LIN {X 0,Y 538.14,Z 616.393,A -85,B 0,C 180,E1 -4151.68,E2 -4151.68} C_VEL
LIN {X 0,Y 538.436,Z 594.869,A -85,B 0,C 180,E1 -4154.665,E2 -4154.665} C_VEL
LIN {X 0,Y 538.828,Z 571.509,A -85,B 0,C 180,E1 -4157.948,E2 -4157.948} C_VEL
LIN {X 0,Y 539.184,Z 551.118,A -85,B 0,C 180,E1 -4160.805,E2 -4160.805} C_VEL
LIN {X 0,Y 539.601,Z 529.757,A -85,B 0,C 180,E1 -4163.813,E2 -4163.813} C_VEL
LIN {X 0,Y 539.337,Z 523.937,A -85,B 0,C 180,E1 -4164.645,E2 -4164.645} C_VEL
LIN {X 0,Y 539.061,Z 522.492,A -85,B 0,C 180,E1 -4164.86,E2 -4164.86} C_VEL
LIN {X 0,Y 537.997,Z 520.573,A -85,B 0,C 180,E1 -4165.217,E2 -4165.217} C_VEL
LIN {X 0,Y 535.449,Z 519.098,A -85,B 0,C 180,E1 -4165.705,E2 -4165.705} C_VEL
LIN {X 0,Y 532.19,Z 518.422,A -85,B 0,C 180,E1 -4166.352,E2 -4166.352} C_VEL
LIN {X 0,Y 531.093,Z 518.344,A -85,B 0,C 180,E1 -4166.774,E2 -4166.774} C_VEL
LIN {X 0,Y 531.002,Z 518.341,A -85,B 0,C 180,E1 -4166.921,E2 -4166.921} C_VEL
LIN {X 0,Y 530.985,Z 518.344,A -85,B 0,C 180,E1 -4169.323,E2 -4169.323} C_VEL
LIN {X 0,Y 530.969,Z 518.345,A -85,B 0,C 180,E1 -4172.1,E2 -4172.1} C_VEL
LIN {X 0,Y 530.987,Z 518.339,A -85,B 0,C 180,E1 -4174.853,E2 -4174.853} C_VEL
LIN {X 0,Y 530.969,Z 518.349,A -85,B 0,C 180,E1 -4177.508,E2 -4177.508} C_VEL
LIN {X 0,Y 530.985,Z 518.333,A -85,B 0,C 180,E1 -4180.433,E2 -4180.433} C_VEL
LIN {X 0,Y 530.952,Z 518.337,A -85,B 0,C 180,E1 -4183.279,E2 -4183.279} C_VEL
LIN {X 0,Y 530.986,Z 518.344,A -85,B 0,C 180,E1 -4185.621,E2 -4185.621} C_VEL
LIN {X 0,Y 530.998,Z 518.336,A -85,B 0,C 180,E1 -4188.564,E2 -4188.564} C_VEL
LIN {X 0,Y 530.961,Z 518.344,A -85,B 0,C 180,E1 -4191.529,E2 -4191.529} C_VEL
LIN {X 0,Y 530.958,Z 518.342,A -85,B 0,C 180,E1 -4194.38,E2 -4194.38} C_VEL
LIN {X 0,Y 530.971,Z 518.349,A -85,B 0,C 180,E1 -4197.133,E2 -4197.133} C_VEL
LIN {X 0,Y 530.974,Z 518.341,A -85,B 0,C 180,E1 -4199.803,E2 -4199.803} C_VEL
LIN {X 0,Y 531.018,Z 518.338,A -85,B 0,C 180,E1 -4202.467,E2 -4202.467} C_VEL
LIN {X 0,Y 530.999,Z 518.342,A -85,B 0,C 180,E1 -4204.942,E2 -4204.942} C_VEL
LIN {X 0,Y 530.977,Z 518.342,A -85,B 0,C 180,E1 -4208.246,E2 -4208.246} C_VEL
LIN {X 0,Y 531.049,Z 518.493,A -85,B 0,C 180,E1 -4209.545,E2 -4209.545} C_VEL
LIN {X 0,Y 531.712,Z 523.2,A -85,B 0,C 180,E1 -4210.505,E2 -4210.505} C_VEL
LIN {X 0,Y 531.398,Z 538.775,A -85,B 0,C 180,E1 -4213.48,E2 -4213.48} C_VEL
LIN {X 0,Y 531.21,Z 547.447,A -85,B 0,C 180,E1 -4215.07,E2 -4215.07} C_VEL
LIN {X 0,Y 531.552,Z 549.947,A -85,B 0,C 180,E1 -4215.153,E2 -4215.153} C_VEL
LIN {X 0,Y 532.79,Z 556.751,A -85,B 0,C 180,E1 -4215.282,E2 -4215.282} C_VEL
LIN {X 0,Y 532.431,Z 654.189,A -85,B 0,C 180,E1 -4216.619,E2 -4216.619} C_VEL
LIN {X 0,Y 532.263,Z 667.4,A -85,B 0,C 180,E1 -4216.955,E2 -4216.955} C_VEL
LIN {X 0,Y 532.009,Z 679.509,A -85,B 0,C 180,E1 -4217.41,E2 -4217.41} C_VEL
LIN {X 0,Y 531.827,Z 691.229,A -85,B 0,C 180,E1 -4218.006,E2 -4218.006} C_VEL
LIN {X 0,Y 531.56,Z 702.618,A -85,B 0,C 180,E1 -4218.754,E2 -4218.754} C_VEL
LIN {X 0,Y 531.28,Z 713.098,A -85,B 0,C 180,E1 -4219.616,E2 -4219.616} C_VEL
LIN {X 0,Y 531.071,Z 721.693,A -85,B 0,C 180,E1 -4220.478,E2 -4220.478} C_VEL
LIN {X 0,Y 530.892,Z 729.61,A -85,B 0,C 180,E1 -4221.435,E2 -4221.435} C_VEL
LIN {X 0,Y 530.69,Z 737.354,A -85,B 0,C 180,E1 -4222.581,E2 -4222.581} C_VEL
LIN {X 0,Y 530.607,Z 744.464,A -85,B 0,C 180,E1 -4223.917,E2 -4223.917} C_VEL
LIN {X 0,Y 530.459,Z 749.203,A -85,B 0,C 180,E1 -4225.059,E2 -4225.059} C_VEL
LIN {X 0,Y 530.516,Z 752.832,A -85,B 0,C 180,E1 -4226.201,E2 -4226.201} C_VEL
LIN {X 0,Y 530.457,Z 754.711,A -85,B 0,C 180,E1 -4226.962,E2 -4226.962} C_VEL
LIN {X 0,Y 530.411,Z 756.13,A -85,B 0,C 180,E1 -4227.721,E2 -4227.721} C_VEL
LIN {X 0,Y 530.344,Z 757.757,A -85,B 0,C 180,E1 -4229.24,E2 -4229.24} C_VEL
LIN {X 0,Y 530.343,Z 757.996,A -85,B 0,C 180,E1 -4229.999,E2 -4229.999} C_VEL
LIN {X 0,Y 530.344,Z 757.814,A -85,B 0,C 180,E1 -4230.759,E2 -4230.759} C_VEL
LIN {X 0,Y 530.411,Z 756.265,A -85,B 0,C 180,E1 -4232.277,E2 -4232.277} C_VEL
LIN {X 0,Y 530.457,Z 754.903,A -85,B 0,C 180,E1 -4233.037,E2 -4233.037} C_VEL
LIN {X 0,Y 530.523,Z 752.021,A -85,B 0,C 180,E1 -4234.178,E2 -4234.178} C_VEL
LIN {X 0,Y 530.523,Z 748.12,A -85,B 0,C 180,E1 -4235.32,E2 -4235.32} C_VEL
LIN {X 0,Y 530.592,Z 742.537,A -85,B 0,C 180,E1 -4236.575,E2 -4236.575} C_VEL
LIN {X 0,Y 530.758,Z 735.529,A -85,B 0,C 180,E1 -4237.8,E2 -4237.8} C_VEL
LIN {X 0,Y 530.927,Z 727.343,A -85,B 0,C 180,E1 -4238.947,E2 -4238.947} C_VEL
LIN {X 0,Y 531.104,Z 718.972,A -85,B 0,C 180,E1 -4239.905,E2 -4239.905} C_VEL
LIN {X 0,Y 531.418,Z 708.669,A -85,B 0,C 180,E1 -4240.862,E2 -4240.862} C_VEL
LIN {X 0,Y 531.692,Z 698.123,A -85,B 0,C 180,E1 -4241.651,E2 -4241.651} C_VEL
LIN {X 0,Y 531.871,Z 687.285,A -85,B 0,C 180,E1 -4242.302,E2 -4242.302} C_VEL
LIN {X 0,Y 532.16,Z 674.779,A -85,B 0,C 180,E1 -4242.876,E2 -4242.876} C_VEL
LIN {X 0,Y 532.357,Z 661.342,A -85,B 0,C 180,E1 -4243.308,E2 -4243.308} C_VEL
LIN {X 0,Y 532.508,Z 647.991,A -85,B 0,C 180,E1 -4243.572,E2 -4243.572} C_VEL
LIN {X 0,Y 532.735,Z 556.433,A -85,B 0,C 180,E1 -4244.814,E2 -4244.814} C_VEL
LIN {X 0,Y 531.26,Z 547.806,A -85,B 0,C 180,E1 -4244.989,E2 -4244.989} C_VEL
LIN {X 0,Y 531.226,Z 545.512,A -85,B 0,C 180,E1 -4245.342,E2 -4245.342} C_VEL
LIN {X 0,Y 531.549,Z 530.014,A -85,B 0,C 180,E1 -4248.281,E2 -4248.281} C_VEL
LIN {X 0,Y 531.675,Z 522.634,A -85,B 0,C 180,E1 -4249.698,E2 -4249.698} C_VEL
LIN {X 0,Y 531.04,Z 518.404,A -85,B 0,C 180,E1 -4250.58,E2 -4250.58} C_VEL
LIN {X 0,Y 530.998,Z 518.339,A -85,B 0,C 180,E1 -4254.042,E2 -4254.042} C_VEL
LIN {X 0,Y 531.006,Z 518.336,A -85,B 0,C 180,E1 -4256.743,E2 -4256.743} C_VEL
LIN {X 0,Y 530.982,Z 518.342,A -85,B 0,C 180,E1 -4259.322,E2 -4259.322} C_VEL
LIN {X 0,Y 530.979,Z 518.34,A -85,B 0,C 180,E1 -4262.102,E2 -4262.102} C_VEL
LIN {X 0,Y 530.987,Z 518.341,A -85,B 0,C 180,E1 -4264.853,E2 -4264.853} C_VEL
LIN {X 0,Y 530.965,Z 518.349,A -85,B 0,C 180,E1 -4267.507,E2 -4267.507} C_VEL
LIN {X 0,Y 530.982,Z 518.336,A -85,B 0,C 180,E1 -4270.432,E2 -4270.432} C_VEL
LIN {X 0,Y 530.968,Z 518.348,A -85,B 0,C 180,E1 -4273.281,E2 -4273.281} C_VEL
LIN {X 0,Y 530.984,Z 518.344,A -85,B 0,C 180,E1 -4275.62,E2 -4275.62} C_VEL
LIN {X 0,Y 531.003,Z 518.336,A -85,B 0,C 180,E1 -4278.565,E2 -4278.565} C_VEL
LIN {X 0,Y 530.964,Z 518.342,A -85,B 0,C 180,E1 -4281.345,E2 -4281.345} C_VEL
LIN {X 0,Y 530.978,Z 518.339,A -85,B 0,C 180,E1 -4284.382,E2 -4284.382} C_VEL
LIN {X 0,Y 530.97,Z 518.344,A -85,B 0,C 180,E1 -4287.133,E2 -4287.133} C_VEL
LIN {X 0,Y 530.981,Z 518.343,A -85,B 0,C 180,E1 -4289.804,E2 -4289.804} C_VEL
LIN {X 0,Y 531.012,Z 518.332,A -85,B 0,C 180,E1 -4292.466,E2 -4292.466} C_VEL
LIN {X 0,Y 531.002,Z 518.338,A -85,B 0,C 180,E1 -4294.942,E2 -4294.942} C_VEL
LIN {X 0,Y 530.965,Z 518.339,A -85,B 0,C 180,E1 -4298.246,E2 -4298.246} C_VEL
LIN {X 0,Y 530.991,Z 518.337,A -85,B 0,C 180,E1 -4300.677,E2 -4300.677} C_VEL
LIN {X 0,Y 530.987,Z 518.339,A -85,B 0,C 180,E1 -4303.071,E2 -4303.071} C_VEL
LIN {X 0,Y 531.012,Z 518.34,A -85,B 0,C 180,E1 -4305.436,E2 -4305.436} C_VEL
LIN {X 0,Y 531.029,Z 518.331,A -85,B 0,C 180,E1 -4308.549,E2 -4308.549} C_VEL
LIN {X 0,Y 531.053,Z 518.337,A -85,B 0,C 180,E1 -4311.629,E2 -4311.629} C_VEL
LIN {X 0,Y 531.117,Z 518.321,A -85,B 0,C 180,E1 -4314.685,E2 -4314.685} C_VEL
LIN {X 0,Y 531.133,Z 518.325,A -85,B 0,C 180,E1 -4317.725,E2 -4317.725} C_VEL
LIN {X 0,Y 531.148,Z 518.318,A -85,B 0,C 180,E1 -4320.758,E2 -4320.758} C_VEL
LIN {X 0,Y 531.102,Z 518.323,A -85,B 0,C 180,E1 -4323.034,E2 -4323.034} C_VEL
LIN {X 0,Y 531.077,Z 518.329,A -85,B 0,C 180,E1 -4326.077,E2 -4326.077} C_VEL
LIN {X 0,Y 531.025,Z 518.335,A -85,B 0,C 180,E1 -4329.138,E2 -4329.138} C_VEL
LIN {X 0,Y 531.033,Z 518.333,A -85,B 0,C 180,E1 -4332.225,E2 -4332.225} C_VEL
LIN {X 0,Y 530.989,Z 518.342,A -85,B 0,C 180,E1 -4335.35,E2 -4335.35} C_VEL
LIN {X 0,Y 531.009,Z 518.343,A -85,B 0,C 180,E1 -4337.723,E2 -4337.723} C_VEL
LIN {X 0,Y 530.995,Z 518.337,A -85,B 0,C 180,E1 -4340.938,E2 -4340.938} C_VEL
LIN {X 0,Y 530.973,Z 518.341,A -85,B 0,C 180,E1 -4344.225,E2 -4344.225} C_VEL
LIN {X 0,Y 531.005,Z 518.333,A -85,B 0,C 180,E1 -4346.744,E2 -4346.744} C_VEL
LIN {X 0,Y 530.976,Z 518.344,A -85,B 0,C 180,E1 -4349.323,E2 -4349.323} C_VEL
LIN {X 0,Y 530.975,Z 518.342,A -85,B 0,C 180,E1 -4352.104,E2 -4352.104} C_VEL
LIN {X 0,Y 530.986,Z 518.337,A -85,B 0,C 180,E1 -4354.855,E2 -4354.855} C_VEL
LIN {X 0,Y 530.961,Z 518.342,A -85,B 0,C 180,E1 -4357.508,E2 -4357.508} C_VEL
LIN {X 0,Y 530.98,Z 518.339,A -85,B 0,C 180,E1 -4360.433,E2 -4360.433} C_VEL
LIN {X 0,Y 530.959,Z 518.341,A -85,B 0,C 180,E1 -4363.282,E2 -4363.282} C_VEL
LIN {X 0,Y 530.984,Z 518.347,A -85,B 0,C 180,E1 -4365.621,E2 -4365.621} C_VEL
LIN {X 0,Y 531.004,Z 518.336,A -85,B 0,C 180,E1 -4368.567,E2 -4368.567} C_VEL
LIN {X 0,Y 530.966,Z 518.342,A -85,B 0,C 180,E1 -4371.347,E2 -4371.347} C_VEL
LIN {X 0,Y 530.974,Z 518.341,A -85,B 0,C 180,E1 -4374.383,E2 -4374.383} C_VEL
LIN {X 0,Y 530.971,Z 518.338,A -85,B 0,C 180,E1 -4377.135,E2 -4377.135} C_VEL
LIN {X 0,Y 530.968,Z 518.329,A -85,B 0,C 180,E1 -4379.804,E2 -4379.804} C_VEL
LIN {X 0,Y 531.015,Z 518.334,A -85,B 0,C 180,E1 -4382.468,E2 -4382.468} C_VEL
LIN {X 0,Y 531.006,Z 518.336,A -85,B 0,C 180,E1 -4384.943,E2 -4384.943} C_VEL
LIN {X 0,Y 531.017,Z 518.525,A -85,B 0,C 180,E1 -4385.967,E2 -4385.967} C_VEL
LIN {X 0,Y 532.382,Z 526.216,A -85,B 0,C 180,E1 -4387.287,E2 -4387.287} C_VEL
LIN {X 0,Y 531.99,Z 544.026,A -85,B 0,C 180,E1 -4390.113,E2 -4390.113} C_VEL
LIN {X 0,Y 531.618,Z 561.828,A -85,B 0,C 180,E1 -4392.895,E2 -4392.895} C_VEL
LIN {X 0,Y 531.386,Z 575.726,A -85,B 0,C 180,E1 -4395.018,E2 -4395.018} C_VEL
LIN {X 0,Y 531.936,Z 579.532,A -85,B 0,C 180,E1 -4395.119,E2 -4395.119} C_VEL
LIN {X 0,Y 532.852,Z 586.518,A -85,B 0,C 180,E1 -4395.24,E2 -4395.24} C_VEL
LIN {X 0,Y 532.462,Z 683.946,A -85,B 0,C 180,E1 -4396.573,E2 -4396.573} C_VEL
LIN {X 0,Y 532.241,Z 697.212,A -85,B 0,C 180,E1 -4396.907,E2 -4396.907} C_VEL
LIN {X 0,Y 532.003,Z 710.498,A -85,B 0,C 180,E1 -4397.411,E2 -4397.411} C_VEL
LIN {X 0,Y 531.803,Z 721.953,A -85,B 0,C 180,E1 -4398.007,E2 -4398.007} C_VEL
LIN {X 0,Y 531.557,Z 733.203,A -85,B 0,C 180,E1 -4398.755,E2 -4398.755} C_VEL
LIN {X 0,Y 531.267,Z 743.612,A -85,B 0,C 180,E1 -4399.617,E2 -4399.617} C_VEL
LIN {X 0,Y 531.06,Z 752.12,A -85,B 0,C 180,E1 -4400.479,E2 -4400.479} C_VEL
LIN {X 0,Y 530.886,Z 759.966,A -85,B 0,C 180,E1 -4401.436,E2 -4401.436} C_VEL
LIN {X 0,Y 530.684,Z 767.626,A -85,B 0,C 180,E1 -4402.582,E2 -4402.582} C_VEL
LIN {X 0,Y 530.603,Z 774.682,A -85,B 0,C 180,E1 -4403.918,E2 -4403.918} C_VEL
LIN {X 0,Y 530.459,Z 779.375,A -85,B 0,C 180,E1 -4405.06,E2 -4405.06} C_VEL
LIN {X 0,Y 530.516,Z 782.962,A -85,B 0,C 180,E1 -4406.203,E2 -4406.203} C_VEL
LIN {X 0,Y 530.457,Z 784.811,A -85,B 0,C 180,E1 -4406.963,E2 -4406.963} C_VEL
LIN {X 0,Y 530.41,Z 786.197,A -85,B 0,C 180,E1 -4407.723,E2 -4407.723} C_VEL
LIN {X 0,Y 530.344,Z 787.786,A -85,B 0,C 180,E1 -4409.241,E2 -4409.241} C_VEL
LIN {X 0,Y 530.342,Z 788,A -85,B 0,C 180,E1 -4410.001,E2 -4410.001} C_VEL
LIN {X 0,Y 530.361,Z 787.182,A -85,B 0,C 180,E1 -4411.519,E2 -4411.519} C_VEL
LIN {X 0,Y 530.41,Z 786.193,A -85,B 0,C 180,E1 -4412.279,E2 -4412.279} C_VEL
LIN {X 0,Y 530.457,Z 784.805,A -85,B 0,C 180,E1 -4413.038,E2 -4413.038} C_VEL
LIN {X 0,Y 530.522,Z 781.892,A -85,B 0,C 180,E1 -4414.179,E2 -4414.179} C_VEL
LIN {X 0,Y 530.525,Z 777.947,A -85,B 0,C 180,E1 -4415.321,E2 -4415.321} C_VEL
LIN {X 0,Y 530.599,Z 772.261,A -85,B 0,C 180,E1 -4416.582,E2 -4416.582} C_VEL
LIN {X 0,Y 530.759,Z 765.231,A -85,B 0,C 180,E1 -4417.801,E2 -4417.801} C_VEL
LIN {X 0,Y 530.931,Z 756.987,A -85,B 0,C 180,E1 -4418.948,E2 -4418.948} C_VEL
LIN {X 0,Y 531.14,Z 748.534,A -85,B 0,C 180,E1 -4419.906,E2 -4419.906} C_VEL
LIN {X 0,Y 531.413,Z 738.084,A -85,B 0,C 180,E1 -4420.863,E2 -4420.863} C_VEL
LIN {X 0,Y 531.694,Z 727.345,A -85,B 0,C 180,E1 -4421.656,E2 -4421.656} C_VEL
LIN {X 0,Y 531.905,Z 716.395,A -85,B 0,C 180,E1 -4422.302,E2 -4422.302} C_VEL
LIN {X 0,Y 532.132,Z 704.753,A -85,B 0,C 180,E1 -4422.83,E2 -4422.83} C_VEL
LIN {X 0,Y 532.333,Z 691.302,A -85,B 0,C 180,E1 -4423.262,E2 -4423.262} C_VEL
LIN {X 0,Y 532.485,Z 678.006,A -85,B 0,C 180,E1 -4423.525,E2 -4423.525} C_VEL
LIN {X 0,Y 532.711,Z 584.398,A -85,B 0,C 180,E1 -4424.793,E2 -4424.793} C_VEL
LIN {X 0,Y 531.371,Z 575.975,A -85,B 0,C 180,E1 -4424.965,E2 -4424.965} C_VEL
LIN {X 0,Y 531.417,Z 570.721,A -85,B 0,C 180,E1 -4425.731,E2 -4425.731} C_VEL
LIN {X 0,Y 531.814,Z 551.642,A -85,B 0,C 180,E1 -4428.692,E2 -4428.692} C_VEL
LIN {X 0,Y 532.238,Z 532.567,A -85,B 0,C 180,E1 -4431.699,E2 -4431.699} C_VEL
LIN {X 0,Y 532.254,Z 524.933,A -85,B 0,C 180,E1 -4432.925,E2 -4432.925} C_VEL
LIN {X 0,Y 531.005,Z 518.517,A -85,B 0,C 180,E1 -4434.043,E2 -4434.043} C_VEL
LIN {X 0,Y 531.009,Z 518.341,A -85,B 0,C 180,E1 -4436.744,E2 -4436.744} C_VEL
LIN {X 0,Y 530.986,Z 518.333,A -85,B 0,C 180,E1 -4439.323,E2 -4439.323} C_VEL
LIN {X 0,Y 530.97,Z 518.348,A -85,B 0,C 180,E1 -4442.101,E2 -4442.101} C_VEL
LIN {X 0,Y 530.974,Z 518.341,A -85,B 0,C 180,E1 -4444.851,E2 -4444.851} C_VEL
LIN {X 0,Y 530.969,Z 518.341,A -85,B 0,C 180,E1 -4447.508,E2 -4447.508} C_VEL
LIN {X 0,Y 530.985,Z 518.345,A -85,B 0,C 180,E1 -4450.433,E2 -4450.433} C_VEL
LIN {X 0,Y 530.969,Z 518.342,A -85,B 0,C 180,E1 -4453.495,E2 -4453.495} C_VEL
LIN {X 0,Y 530.958,Z 518.348,A -85,B 0,C 180,E1 -4456.504,E2 -4456.504} C_VEL
LIN {X 0,Y 530.987,Z 518.339,A -85,B 0,C 180,E1 -4458.977,E2 -4458.977} C_VEL
LIN {X 0,Y 530.961,Z 518.343,A -85,B 0,C 180,E1 -4461.53,E2 -4461.53} C_VEL
LIN {X 0,Y 530.98,Z 518.346,A -85,B 0,C 180,E1 -4464.382,E2 -4464.382} C_VEL
LIN {X 0,Y 530.97,Z 518.341,A -85,B 0,C 180,E1 -4467.133,E2 -4467.133} C_VEL
LIN {X 0,Y 530.973,Z 518.346,A -85,B 0,C 180,E1 -4469.803,E2 -4469.803} C_VEL
LIN {X 0,Y 531.019,Z 518.342,A -85,B 0,C 180,E1 -4472.467,E2 -4472.467} C_VEL
LIN {X 0,Y 531.074,Z 518.473,A -85,B 0,C 180,E1 -4474.658,E2 -4474.658} C_VEL
LIN {X 0,Y 532.431,Z 526.751,A -85,B 0,C 180,E1 -4475.846,E2 -4475.846} C_VEL
LIN {X 0,Y 532.151,Z 548.016,A -85,B 0,C 180,E1 -4478.704,E2 -4478.704} C_VEL
LIN {X 0,Y 531.897,Z 565.291,A -85,B 0,C 180,E1 -4481.112,E2 -4481.112} C_VEL
LIN {X 0,Y 531.698,Z 578.244,A -85,B 0,C 180,E1 -4482.896,E2 -4482.896} C_VEL
LIN {X 0,Y 531.337,Z 598.983,A -85,B 0,C 180,E1 -4485.836,E2 -4485.836} C_VEL
LIN {X 0,Y 531.125,Z 616.376,A -85,B 0,C 180,E1 -4488.252,E2 -4488.252} C_VEL
LIN {X 0,Y 531.903,Z 624.421,A -85,B 0,C 180,E1 -4488.404,E2 -4488.404} C_VEL
LIN {X 0,Y 531.735,Z 695.869,A -85,B 0,C 180,E1 -4489.385,E2 -4489.385} C_VEL
LIN {X 0,Y 531.597,Z 706.827,A -85,B 0,C 180,E1 -4489.671,E2 -4489.671} C_VEL
LIN {X 0,Y 531.429,Z 717.65,A -85,B 0,C 180,E1 -4490.1,E2 -4490.1} C_VEL
LIN {X 0,Y 531.259,Z 728.113,A -85,B 0,C 180,E1 -4490.674,E2 -4490.674} C_VEL
LIN {X 0,Y 531.084,Z 737.485,A -85,B 0,C 180,E1 -4491.342,E2 -4491.342} C_VEL
LIN {X 0,Y 530.882,Z 746.887,A -85,B 0,C 180,E1 -4492.201,E2 -4492.201} C_VEL
LIN {X 0,Y 530.759,Z 755.07,A -85,B 0,C 180,E1 -4493.156,E2 -4493.156} C_VEL
LIN {X 0,Y 530.717,Z 761.555,A -85,B 0,C 180,E1 -4494.109,E2 -4494.109} C_VEL
LIN {X 0,Y 530.513,Z 766.732,A -85,B 0,C 180,E1 -4495.06,E2 -4495.06} C_VEL
LIN {X 0,Y 530.527,Z 771.465,A -85,B 0,C 180,E1 -4496.202,E2 -4496.202} C_VEL
LIN {X 0,Y 530.471,Z 773.822,A -85,B 0,C 180,E1 -4496.962,E2 -4496.962} C_VEL
LIN {X 0,Y 530.411,Z 775.621,A -85,B 0,C 180,E1 -4497.722,E2 -4497.722} C_VEL
LIN {X 0,Y 530.359,Z 776.913,A -85,B 0,C 180,E1 -4498.481,E2 -4498.481} C_VEL
LIN {X 0,Y 530.341,Z 777.704,A -85,B 0,C 180,E1 -4499.241,E2 -4499.241} C_VEL
LIN {X 0,Y 530.341,Z 777.997,A -85,B 0,C 180,E1 -4500,E2 -4500} C_VEL
LIN {X 0,Y 530.342,Z 777.777,A -85,B 0,C 180,E1 -4500.759,E2 -4500.759} C_VEL
LIN {X 0,Y 530.362,Z 777.041,A -85,B 0,C 180,E1 -4501.519,E2 -4501.519} C_VEL
LIN {X 0,Y 530.412,Z 775.802,A -85,B 0,C 180,E1 -4502.278,E2 -4502.278} C_VEL
LIN {X 0,Y 530.497,Z 772.985,A -85,B 0,C 180,E1 -4503.418,E2 -4503.418} C_VEL
LIN {X 0,Y 530.506,Z 768.863,A -85,B 0,C 180,E1 -4504.559,E2 -4504.559} C_VEL
LIN {X 0,Y 530.658,Z 763.231,A -85,B 0,C 180,E1 -4505.701,E2 -4505.701} C_VEL
LIN {X 0,Y 530.713,Z 756.929,A -85,B 0,C 180,E1 -4506.688,E2 -4506.688} C_VEL
LIN {X 0,Y 530.841,Z 749.531,A -85,B 0,C 180,E1 -4507.608,E2 -4507.608} C_VEL
LIN {X 0,Y 531.011,Z 740.852,A -85,B 0,C 180,E1 -4508.467,E2 -4508.467} C_VEL
LIN {X 0,Y 531.278,Z 730.982,A -85,B 0,C 180,E1 -4509.23,E2 -4509.23} C_VEL
LIN {X 0,Y 531.391,Z 721.423,A -85,B 0,C 180,E1 -4509.804,E2 -4509.804} C_VEL
LIN {X 0,Y 531.569,Z 710.783,A -85,B 0,C 180,E1 -4510.282,E2 -4510.282} C_VEL
LIN {X 0,Y 531.674,Z 699.003,A -85,B 0,C 180,E1 -4510.641,E2 -4510.641} C_VEL
LIN {X 0,Y 531.79,Z 684.449,A -85,B 0,C 180,E1 -4510.879,E2 -4510.879} C_VEL
LIN {X 0,Y 531.778,Z 622.376,A -85,B 0,C 180,E1 -4511.717,E2 -4511.717} C_VEL
LIN {X 0,Y 531.114,Z 616.427,A -85,B 0,C 180,E1 -4511.834,E2 -4511.834} C_VEL
LIN {X 0,Y 531.456,Z 594.899,A -85,B 0,C 180,E1 -4514.839,E2 -4514.839} C_VEL
LIN {X 0,Y 531.89,Z 570.346,A -85,B 0,C 180,E1 -4518.314,E2 -4518.314} C_VEL
LIN {X 0,Y 532.269,Z 549.336,A -85,B 0,C 180,E1 -4521.291,E2 -4521.291} C_VEL
LIN {X 0,Y 532.648,Z 529.254,A -85,B 0,C 180,E1 -4524.144,E2 -4524.144} C_VEL
LIN {X 0,Y 532.198,Z 524.25,A -85,B 0,C 180,E1 -4524.876,E2 -4524.876} C_VEL
LIN {X 0,Y 531.025,Z 518.439,A -85,B 0,C 180,E1 -4525.797,E2 -4525.797} C_VEL
LIN {X 0,Y 531.002,Z 518.341,A -85,B 0,C 180,E1 -4526.921,E2 -4526.921} C_VEL
LIN {X 0,Y 530.327,Z 518.429,A -85,B 0,C 180,E1 -4527.554,E2 -4527.554} C_VEL
LIN {X 0,Y 527.455,Z 518.785,A -85,B 0,C 180,E1 -4528.582,E2 -4528.582} C_VEL
LIN {X 0,Y 525.039,Z 519.086,A -85,B 0,C 180,E1 -4529.409,E2 -4529.409} C_VEL
LIN {X 0,Y 524.014,Z 519.213,A -85,B 0,C 180,E1 -4530.049,E2 -4530.049} C_VEL
LIN {X 0,Y 523.938,Z 519.219,A -85,B 0,C 180,E1 -4530.265,E2 -4530.265} C_VEL
LIN {X 0,Y 523.945,Z 519.221,A -85,B 0,C 180,E1 -4533.364,E2 -4533.364} C_VEL
LIN {X 0,Y 523.911,Z 519.22,A -85,B 0,C 180,E1 -4536.402,E2 -4536.402} C_VEL
LIN {X 0,Y 523.925,Z 519.22,A -85,B 0,C 180,E1 -4539.085,E2 -4539.085} C_VEL
LIN {X 0,Y 523.954,Z 519.201,A -85,B 0,C 180,E1 -4542.119,E2 -4542.119} C_VEL
LIN {X 0,Y 523.95,Z 519.22,A -85,B 0,C 180,E1 -4545.31,E2 -4545.31} C_VEL
LIN {X 0,Y 523.961,Z 519.213,A -85,B 0,C 180,E1 -4548.69,E2 -4548.69} C_VEL
LIN {X 0,Y 523.92,Z 519.218,A -85,B 0,C 180,E1 -4551.898,E2 -4551.898} C_VEL
LIN {X 0,Y 523.928,Z 519.224,A -85,B 0,C 180,E1 -4554.911,E2 -4554.911} C_VEL
LIN {X 0,Y 523.939,Z 519.218,A -85,B 0,C 180,E1 -4557.68,E2 -4557.68} C_VEL
LIN {X 0,Y 523.959,Z 519.22,A -85,B 0,C 180,E1 -4560.676,E2 -4560.676} C_VEL
LIN {X 0,Y 523.978,Z 519.213,A -85,B 0,C 180,E1 -4563.728,E2 -4563.728} C_VEL
LIN {X 0,Y 523.917,Z 519.219,A -85,B 0,C 180,E1 -4566.269,E2 -4566.269} C_VEL
LIN {X 0,Y 523.992,Z 519.334,A -85,B 0,C 180,E1 -4569.385,E2 -4569.385} C_VEL
LIN {X 0,Y 524.768,Z 524.408,A -85,B 0,C 180,E1 -4570.438,E2 -4570.438} C_VEL
LIN {X 0,Y 524.356,Z 541.047,A -85,B 0,C 180,E1 -4573.652,E2 -4573.652} C_VEL
LIN {X 0,Y 524.229,Z 547.516,A -85,B 0,C 180,E1 -4574.854,E2 -4574.854} C_VEL
LIN {X 0,Y 524.588,Z 550.04,A -85,B 0,C 180,E1 -4574.949,E2 -4574.949} C_VEL
LIN {X 0,Y 525.943,Z 557.681,A -85,B 0,C 180,E1 -4575.096,E2 -4575.096} C_VEL
LIN {X 0,Y 525.546,Z 654.422,A -85,B 0,C 180,E1 -4576.441,E2 -4576.441} C_VEL
LIN {X 0,Y 525.372,Z 667.622,A -85,B 0,C 180,E1 -4576.781,E2 -4576.781} C_VEL
LIN {X 0,Y 525.105,Z 679.724,A -85,B 0,C 180,E1 -4577.241,E2 -4577.241} C_VEL
LIN {X 0,Y 524.901,Z 690.664,A -85,B 0,C 180,E1 -4577.8,E2 -4577.8} C_VEL
LIN {X 0,Y 524.651,Z 701.514,A -85,B 0,C 180,E1 -4578.506,E2 -4578.506} C_VEL
LIN {X 0,Y 524.319,Z 712.217,A -85,B 0,C 180,E1 -4579.379,E2 -4579.379} C_VEL
LIN {X 0,Y 524.061,Z 721.842,A -85,B 0,C 180,E1 -4580.349,E2 -4580.349} C_VEL
LIN {X 0,Y 523.86,Z 729.724,A -85,B 0,C 180,E1 -4581.319,E2 -4581.319} C_VEL
LIN {X 0,Y 523.637,Z 737.431,A -85,B 0,C 180,E1 -4582.48,E2 -4582.48} C_VEL
LIN {X 0,Y 523.519,Z 744.5,A -85,B 0,C 180,E1 -4583.834,E2 -4583.834} C_VEL
LIN {X 0,Y 523.384,Z 749.231,A -85,B 0,C 180,E1 -4584.992,E2 -4584.992} C_VEL
LIN {X 0,Y 523.444,Z 752.84,A -85,B 0,C 180,E1 -4586.15,E2 -4586.15} C_VEL
LIN {X 0,Y 523.368,Z 754.712,A -85,B 0,C 180,E1 -4586.92,E2 -4586.92} C_VEL
LIN {X 0,Y 523.335,Z 756.13,A -85,B 0,C 180,E1 -4587.69,E2 -4587.69} C_VEL
LIN {X 0,Y 523.25,Z 757.757,A -85,B 0,C 180,E1 -4589.23,E2 -4589.23} C_VEL
LIN {X 0,Y 523.247,Z 757.997,A -85,B 0,C 180,E1 -4589.999,E2 -4589.999} C_VEL
LIN {X 0,Y 523.25,Z 757.814,A -85,B 0,C 180,E1 -4590.769,E2 -4590.769} C_VEL
LIN {X 0,Y 523.335,Z 756.263,A -85,B 0,C 180,E1 -4592.308,E2 -4592.308} C_VEL
LIN {X 0,Y 523.368,Z 754.901,A -85,B 0,C 180,E1 -4593.078,E2 -4593.078} C_VEL
LIN {X 0,Y 523.442,Z 752.025,A -85,B 0,C 180,E1 -4594.234,E2 -4594.234} C_VEL
LIN {X 0,Y 523.462,Z 748.133,A -85,B 0,C 180,E1 -4595.392,E2 -4595.392} C_VEL
LIN {X 0,Y 523.516,Z 743.024,A -85,B 0,C 180,E1 -4596.574,E2 -4596.574} C_VEL
LIN {X 0,Y 523.664,Z 736.829,A -85,B 0,C 180,E1 -4597.712,E2 -4597.712} C_VEL
LIN {X 0,Y 523.876,Z 728.94,A -85,B 0,C 180,E1 -4598.874,E2 -4598.874} C_VEL
LIN {X 0,Y 524.097,Z 719.123,A -85,B 0,C 180,E1 -4600.039,E2 -4600.039} C_VEL
LIN {X 0,Y 524.444,Z 708.833,A -85,B 0,C 180,E1 -4601.008,E2 -4601.008} C_VEL
LIN {X 0,Y 524.725,Z 698.74,A -85,B 0,C 180,E1 -4601.778,E2 -4601.778} C_VEL
LIN {X 0,Y 524.942,Z 687.481,A -85,B 0,C 180,E1 -4602.467,E2 -4602.467} C_VEL
LIN {X 0,Y 525.257,Z 674.959,A -85,B 0,C 180,E1 -4603.049,E2 -4603.049} C_VEL
LIN {X 0,Y 525.473,Z 661.52,A -85,B 0,C 180,E1 -4603.486,E2 -4603.486} C_VEL
LIN {X 0,Y 525.636,Z 648.151,A -85,B 0,C 180,E1 -4603.753,E2 -4603.753} C_VEL
LIN {X 0,Y 525.881,Z 557.209,A -85,B 0,C 180,E1 -4605.003,E2 -4605.003} C_VEL
LIN {X 0,Y 524.28,Z 547.868,A -85,B 0,C 180,E1 -4605.205,E2 -4605.205} C_VEL
LIN {X 0,Y 524.223,Z 545.692,A -85,B 0,C 180,E1 -4605.552,E2 -4605.552} C_VEL
LIN {X 0,Y 524.583,Z 531.328,A -85,B 0,C 180,E1 -4608.31,E2 -4608.31} C_VEL
LIN {X 0,Y 524.636,Z 523.164,A -85,B 0,C 180,E1 -4609.902,E2 -4609.902} C_VEL
LIN {X 0,Y 523.979,Z 519.256,A -85,B 0,C 180,E1 -4610.742,E2 -4610.742} C_VEL
LIN {X 0,Y 523.963,Z 519.215,A -85,B 0,C 180,E1 -4614.203,E2 -4614.203} C_VEL
LIN {X 0,Y 523.953,Z 519.218,A -85,B 0,C 180,E1 -4617.132,E2 -4617.132} C_VEL
LIN {X 0,Y 523.942,Z 519.218,A -85,B 0,C 180,E1 -4619.755,E2 -4619.755} C_VEL
LIN {X 0,Y 523.939,Z 519.216,A -85,B 0,C 180,E1 -4622.448,E2 -4622.448} C_VEL
LIN {X 0,Y 523.934,Z 519.224,A -85,B 0,C 180,E1 -4625.224,E2 -4625.224} C_VEL
LIN {X 0,Y 523.915,Z 519.22,A -85,B 0,C 180,E1 -4628.101,E2 -4628.101} C_VEL
LIN {X 0,Y 523.959,Z 519.219,A -85,B 0,C 180,E1 -4631.31,E2 -4631.31} C_VEL
LIN {X 0,Y 523.952,Z 519.211,A -85,B 0,C 180,E1 -4634.691,E2 -4634.691} C_VEL
LIN {X 0,Y 523.953,Z 519.217,A -85,B 0,C 180,E1 -4637.881,E2 -4637.881} C_VEL
LIN {X 0,Y 523.955,Z 519.212,A -85,B 0,C 180,E1 -4640.918,E2 -4640.918} C_VEL
LIN {X 0,Y 523.925,Z 519.221,A -85,B 0,C 180,E1 -4643.827,E2 -4643.827} C_VEL
LIN {X 0,Y 523.939,Z 519.216,A -85,B 0,C 180,E1 -4646.635,E2 -4646.635} C_VEL
LIN {X 0,Y 523.958,Z 519.22,A -85,B 0,C 180,E1 -4649.356,E2 -4649.356} C_VEL
LIN {X 0,Y 523.974,Z 519.209,A -85,B 0,C 180,E1 -4652.28,E2 -4652.28} C_VEL
LIN {X 0,Y 523.949,Z 519.214,A -85,B 0,C 180,E1 -4654.581,E2 -4654.581} C_VEL
LIN {X 0,Y 523.91,Z 519.222,A -85,B 0,C 180,E1 -4657.106,E2 -4657.106} C_VEL
LIN {X 0,Y 523.972,Z 519.215,A -85,B 0,C 180,E1 -4659.865,E2 -4659.865} C_VEL
LIN {X 0,Y 523.964,Z 519.212,A -85,B 0,C 180,E1 -4662.837,E2 -4662.837} C_VEL
LIN {X 0,Y 523.969,Z 519.214,A -85,B 0,C 180,E1 -4665.235,E2 -4665.235} C_VEL
LIN {X 0,Y 524.004,Z 519.206,A -85,B 0,C 180,E1 -4668.394,E2 -4668.394} C_VEL
LIN {X 0,Y 524,Z 519.214,A -85,B 0,C 180,E1 -4671.516,E2 -4671.516} C_VEL
LIN {X 0,Y 524.078,Z 519.198,A -85,B 0,C 180,E1 -4674.614,E2 -4674.614} C_VEL
LIN {X 0,Y 524.105,Z 519.201,A -85,B 0,C 180,E1 -4677.694,E2 -4677.694} C_VEL
LIN {X 0,Y 524.118,Z 519.194,A -85,B 0,C 180,E1 -4680.768,E2 -4680.768} C_VEL
LIN {X 0,Y 524.069,Z 519.2,A -85,B 0,C 180,E1 -4683.075,E2 -4683.075} C_VEL
LIN {X 0,Y 524.039,Z 519.205,A -85,B 0,C 180,E1 -4686.159,E2 -4686.159} C_VEL
LIN {X 0,Y 523.993,Z 519.212,A -85,B 0,C 180,E1 -4689.262,E2 -4689.262} C_VEL
LIN {X 0,Y 524.017,Z 519.213,A -85,B 0,C 180,E1 -4691.751,E2 -4691.751} C_VEL
LIN {X 0,Y 523.985,Z 519.211,A -85,B 0,C 180,E1 -4695.053,E2 -4695.053} C_VEL
LIN {X 0,Y 523.957,Z 519.217,A -85,B 0,C 180,E1 -4697.969,E2 -4697.969} C_VEL
LIN {X 0,Y 523.966,Z 519.212,A -85,B 0,C 180,E1 -4700.41,E2 -4700.41} C_VEL
LIN {X 0,Y 523.91,Z 519.219,A -85,B 0,C 180,E1 -4702.894,E2 -4702.894} C_VEL
LIN {X 0,Y 523.949,Z 519.221,A -85,B 0,C 180,E1 -4705.419,E2 -4705.419} C_VEL
LIN {X 0,Y 523.964,Z 519.217,A -85,B 0,C 180,E1 -4707.999,E2 -4707.999} C_VEL
LIN {X 0,Y 523.941,Z 519.215,A -85,B 0,C 180,E1 -4710.856,E2 -4710.856} C_VEL
LIN {X 0,Y 523.957,Z 519.22,A -85,B 0,C 180,E1 -4713.736,E2 -4713.736} C_VEL
LIN {X 0,Y 523.917,Z 519.212,A -85,B 0,C 180,E1 -4716.405,E2 -4716.405} C_VEL
LIN {X 0,Y 523.918,Z 519.22,A -85,B 0,C 180,E1 -4719.085,E2 -4719.085} C_VEL
LIN {X 0,Y 523.952,Z 519.213,A -85,B 0,C 180,E1 -4722.119,E2 -4722.119} C_VEL
LIN {X 0,Y 523.952,Z 519.218,A -85,B 0,C 180,E1 -4725.309,E2 -4725.309} C_VEL
LIN {X 0,Y 523.969,Z 519.213,A -85,B 0,C 180,E1 -4728.688,E2 -4728.688} C_VEL
LIN {X 0,Y 523.923,Z 519.217,A -85,B 0,C 180,E1 -4731.08,E2 -4731.08} C_VEL
LIN {X 0,Y 523.922,Z 519.225,A -85,B 0,C 180,E1 -4733.828,E2 -4733.828} C_VEL
LIN {X 0,Y 523.941,Z 519.211,A -85,B 0,C 180,E1 -4736.637,E2 -4736.637} C_VEL
LIN {X 0,Y 523.955,Z 519.193,A -85,B 0,C 180,E1 -4739.357,E2 -4739.357} C_VEL
LIN {X 0,Y 523.978,Z 519.212,A -85,B 0,C 180,E1 -4742.282,E2 -4742.282} C_VEL
LIN {X 0,Y 523.952,Z 519.208,A -85,B 0,C 180,E1 -4744.582,E2 -4744.582} C_VEL
LIN {X 0,Y 523.986,Z 519.388,A -85,B 0,C 180,E1 -4745.791,E2 -4745.791} C_VEL
LIN {X 0,Y 525.428,Z 527.311,A -85,B 0,C 180,E1 -4747.177,E2 -4747.177} C_VEL
LIN {X 0,Y 525.026,Z 545.12,A -85,B 0,C 180,E1 -4750.042,E2 -4750.042} C_VEL
LIN {X 0,Y 524.582,Z 562.914,A -85,B 0,C 180,E1 -4752.859,E2 -4752.859} C_VEL
LIN {X 0,Y 524.338,Z 575.501,A -85,B 0,C 180,E1 -4754.81,E2 -4754.81} C_VEL
LIN {X 0,Y 524.822,Z 578.883,A -85,B 0,C 180,E1 -4754.906,E2 -4754.906} C_VEL
LIN {X 0,Y 525.978,Z 587.161,A -85,B 0,C 180,E1 -4755.054,E2 -4755.054} C_VEL
LIN {X 0,Y 525.563,Z 683.741,A -85,B 0,C 180,E1 -4756.393,E2 -4756.393} C_VEL
LIN {X 0,Y 525.313,Z 697.006,A -85,B 0,C 180,E1 -4756.731,E2 -4756.731} C_VEL
LIN {X 0,Y 525.054,Z 710.298,A -85,B 0,C 180,E1 -4757.241,E2 -4757.241} C_VEL
LIN {X 0,Y 524.815,Z 722.77,A -85,B 0,C 180,E1 -4757.906,E2 -4757.906} C_VEL
LIN {X 0,Y 524.537,Z 734.361,A -85,B 0,C 180,E1 -4758.7,E2 -4758.7} C_VEL
LIN {X 0,Y 524.244,Z 744.556,A -85,B 0,C 180,E1 -4759.574,E2 -4759.574} C_VEL
LIN {X 0,Y 523.975,Z 753.733,A -85,B 0,C 180,E1 -4760.544,E2 -4760.544} C_VEL
LIN {X 0,Y 523.759,Z 762.675,A -85,B 0,C 180,E1 -4761.707,E2 -4761.707} C_VEL
LIN {X 0,Y 523.583,Z 769.853,A -85,B 0,C 180,E1 -4762.868,E2 -4762.868} C_VEL
LIN {X 0,Y 523.543,Z 776.367,A -85,B 0,C 180,E1 -4764.222,E2 -4764.222} C_VEL
LIN {X 0,Y 523.361,Z 780.679,A -85,B 0,C 180,E1 -4765.379,E2 -4765.379} C_VEL
LIN {X 0,Y 523.443,Z 782.962,A -85,B 0,C 180,E1 -4766.151,E2 -4766.151} C_VEL
LIN {X 0,Y 523.367,Z 784.811,A -85,B 0,C 180,E1 -4766.922,E2 -4766.922} C_VEL
LIN {X 0,Y 523.334,Z 786.197,A -85,B 0,C 180,E1 -4767.692,E2 -4767.692} C_VEL
LIN {X 0,Y 523.25,Z 787.786,A -85,B 0,C 180,E1 -4769.231,E2 -4769.231} C_VEL
LIN {X 0,Y 523.246,Z 788,A -85,B 0,C 180,E1 -4770.001,E2 -4770.001} C_VEL
LIN {X 0,Y 523.274,Z 787.181,A -85,B 0,C 180,E1 -4771.54,E2 -4771.54} C_VEL
LIN {X 0,Y 523.334,Z 786.192,A -85,B 0,C 180,E1 -4772.31,E2 -4772.31} C_VEL
LIN {X 0,Y 523.368,Z 784.805,A -85,B 0,C 180,E1 -4773.08,E2 -4773.08} C_VEL
LIN {X 0,Y 523.441,Z 781.892,A -85,B 0,C 180,E1 -4774.236,E2 -4774.236} C_VEL
LIN {X 0,Y 523.464,Z 777.947,A -85,B 0,C 180,E1 -4775.393,E2 -4775.393} C_VEL
LIN {X 0,Y 523.524,Z 772.725,A -85,B 0,C 180,E1 -4776.581,E2 -4776.581} C_VEL
LIN {X 0,Y 523.665,Z 766.46,A -85,B 0,C 180,E1 -4777.713,E2 -4777.713} C_VEL
LIN {X 0,Y 523.854,Z 758.435,A -85,B 0,C 180,E1 -4778.876,E2 -4778.876} C_VEL
LIN {X 0,Y 524.08,Z 750.253,A -85,B 0,C 180,E1 -4779.845,E2 -4779.845} C_VEL
LIN {X 0,Y 524.355,Z 740.278,A -85,B 0,C 180,E1 -4780.816,E2 -4780.816} C_VEL
LIN {X 0,Y 524.665,Z 729.022,A -85,B 0,C 180,E1 -4781.689,E2 -4781.689} C_VEL
LIN {X 0,Y 524.915,Z 717.979,A -85,B 0,C 180,E1 -4782.37,E2 -4782.37} C_VEL
LIN {X 0,Y 525.153,Z 705.758,A -85,B 0,C 180,E1 -4782.954,E2 -4782.954} C_VEL
LIN {X 0,Y 525.393,Z 692.931,A -85,B 0,C 180,E1 -4783.391,E2 -4783.391} C_VEL
LIN {X 0,Y 525.573,Z 679.321,A -85,B 0,C 180,E1 -4783.682,E2 -4783.682} C_VEL
LIN {X 0,Y 525.891,Z 585.515,A -85,B 0,C 180,E1 -4784.971,E2 -4784.971} C_VEL
LIN {X 0,Y 524.351,Z 575.824,A -85,B 0,C 180,E1 -4785.167,E2 -4785.167} C_VEL
LIN {X 0,Y 524.387,Z 571.792,A -85,B 0,C 180,E1 -4785.748,E2 -4785.748} C_VEL
LIN {X 0,Y 524.83,Z 552.733,A -85,B 0,C 180,E1 -4788.747,E2 -4788.747} C_VEL
LIN {X 0,Y 525.281,Z 533.666,A -85,B 0,C 180,E1 -4791.795,E2 -4791.795} C_VEL
LIN {X 0,Y 525.464,Z 527.31,A -85,B 0,C 180,E1 -4792.823,E2 -4792.823} C_VEL
LIN {X 0,Y 523.977,Z 519.355,A -85,B 0,C 180,E1 -4794.228,E2 -4794.228} C_VEL
LIN {X 0,Y 523.957,Z 519.217,A -85,B 0,C 180,E1 -4797.133,E2 -4797.133} C_VEL
LIN {X 0,Y 523.946,Z 519.212,A -85,B 0,C 180,E1 -4799.756,E2 -4799.756} C_VEL
LIN {X 0,Y 523.937,Z 519.223,A -85,B 0,C 180,E1 -4802.45,E2 -4802.45} C_VEL
LIN {X 0,Y 523.924,Z 519.218,A -85,B 0,C 180,E1 -4805.227,E2 -4805.227} C_VEL
LIN {X 0,Y 523.919,Z 519.226,A -85,B 0,C 180,E1 -4808.102,E2 -4808.102} C_VEL
LIN {X 0,Y 523.944,Z 519.217,A -85,B 0,C 180,E1 -4811.092,E2 -4811.092} C_VEL
LIN {X 0,Y 523.941,Z 519.223,A -85,B 0,C 180,E1 -4814.228,E2 -4814.228} C_VEL
LIN {X 0,Y 523.92,Z 519.221,A -85,B 0,C 180,E1 -4816.833,E2 -4816.833} C_VEL
LIN {X 0,Y 523.942,Z 519.217,A -85,B 0,C 180,E1 -4818.908,E2 -4818.908} C_VEL
LIN {X 0,Y 523.919,Z 519.224,A -85,B 0,C 180,E1 -4821.898,E2 -4821.898} C_VEL
LIN {X 0,Y 523.939,Z 519.218,A -85,B 0,C 180,E1 -4824.91,E2 -4824.91} C_VEL
LIN {X 0,Y 523.938,Z 519.22,A -85,B 0,C 180,E1 -4827.68,E2 -4827.68} C_VEL
LIN {X 0,Y 523.958,Z 519.22,A -85,B 0,C 180,E1 -4830.677,E2 -4830.677} C_VEL
LIN {X 0,Y 523.978,Z 519.219,A -85,B 0,C 180,E1 -4833.729,E2 -4833.729} C_VEL
LIN {X 0,Y 524.049,Z 519.411,A -85,B 0,C 180,E1 -4834.564,E2 -4834.564} C_VEL
LIN {X 0,Y 525.426,Z 527.421,A -85,B 0,C 180,E1 -4835.713,E2 -4835.713} C_VEL
LIN {X 0,Y 525.193,Z 547.247,A -85,B 0,C 180,E1 -4838.408,E2 -4838.408} C_VEL
LIN {X 0,Y 524.895,Z 566.283,A -85,B 0,C 180,E1 -4841.053,E2 -4841.053} C_VEL
LIN {X 0,Y 524.671,Z 580.788,A -85,B 0,C 180,E1 -4843.062,E2 -4843.062} C_VEL
LIN {X 0,Y 524.311,Z 600.143,A -85,B 0,C 180,E1 -4845.84,E2 -4845.84} C_VEL
LIN {X 0,Y 524.101,Z 615.984,A -85,B 0,C 180,E1 -4848.045,E2 -4848.045} C_VEL
LIN {X 0,Y 524.142,Z 616.961,A -85,B 0,C 180,E1 -4848.125,E2 -4848.125} C_VEL
LIN {X 0,Y 524.945,Z 626.086,A -85,B 0,C 180,E1 -4848.28,E2 -4848.28} C_VEL
LIN {X 0,Y 524.769,Z 695.389,A -85,B 0,C 180,E1 -4849.242,E2 -4849.242} C_VEL
LIN {X 0,Y 524.634,Z 706.556,A -85,B 0,C 180,E1 -4849.532,E2 -4849.532} C_VEL
LIN {X 0,Y 524.447,Z 717.503,A -85,B 0,C 180,E1 -4849.967,E2 -4849.967} C_VEL
LIN {X 0,Y 524.242,Z 728.034,A -85,B 0,C 180,E1 -4850.548,E2 -4850.548} C_VEL
LIN {X 0,Y 524.059,Z 737.441,A -85,B 0,C 180,E1 -4851.225,E2 -4851.225} C_VEL
LIN {X 0,Y 523.858,Z 746.873,A -85,B 0,C 180,E1 -4852.096,E2 -4852.096} C_VEL
LIN {X 0,Y 523.698,Z 755.073,A -85,B 0,C 180,E1 -4853.063,E2 -4853.063} C_VEL
LIN {X 0,Y 523.644,Z 761.558,A -85,B 0,C 180,E1 -4854.03,E2 -4854.03} C_VEL
LIN {X 0,Y 523.431,Z 766.733,A -85,B 0,C 180,E1 -4854.993,E2 -4854.993} C_VEL
LIN {X 0,Y 523.456,Z 771.467,A -85,B 0,C 180,E1 -4856.151,E2 -4856.151} C_VEL
LIN {X 0,Y 523.382,Z 773.82,A -85,B 0,C 180,E1 -4856.921,E2 -4856.921} C_VEL
LIN {X 0,Y 523.336,Z 775.623,A -85,B 0,C 180,E1 -4857.691,E2 -4857.691} C_VEL
LIN {X 0,Y 523.273,Z 776.912,A -85,B 0,C 180,E1 -4858.461,E2 -4858.461} C_VEL
LIN {X 0,Y 523.247,Z 777.702,A -85,B 0,C 180,E1 -4859.23,E2 -4859.23} C_VEL
LIN {X 0,Y 523.244,Z 777.997,A -85,B 0,C 180,E1 -4860,E2 -4860} C_VEL
LIN {X 0,Y 523.249,Z 777.776,A -85,B 0,C 180,E1 -4860.77,E2 -4860.77} C_VEL
LIN {X 0,Y 523.275,Z 777.039,A -85,B 0,C 180,E1 -4861.539,E2 -4861.539} C_VEL
LIN {X 0,Y 523.337,Z 775.802,A -85,B 0,C 180,E1 -4862.309,E2 -4862.309} C_VEL
LIN {X 0,Y 523.409,Z 772.983,A -85,B 0,C 180,E1 -4863.464,E2 -4863.464} C_VEL
LIN {X 0,Y 523.409,Z 768.861,A -85,B 0,C 180,E1 -4864.621,E2 -4864.621} C_VEL
LIN {X 0,Y 523.606,Z 763.227,A -85,B 0,C 180,E1 -4865.778,E2 -4865.778} C_VEL
LIN {X 0,Y 523.662,Z 755.749,A -85,B 0,C 180,E1 -4866.938,E2 -4866.938} C_VEL
LIN {X 0,Y 523.849,Z 747.717,A -85,B 0,C 180,E1 -4867.904,E2 -4867.904} C_VEL
LIN {X 0,Y 524.06,Z 738.515,A -85,B 0,C 180,E1 -4868.775,E2 -4868.775} C_VEL
LIN {X 0,Y 524.238,Z 729.42,A -85,B 0,C 180,E1 -4869.452,E2 -4869.452} C_VEL
LIN {X 0,Y 524.417,Z 719.348,A -85,B 0,C 180,E1 -4870.033,E2 -4870.033} C_VEL
LIN {X 0,Y 524.606,Z 707.782,A -85,B 0,C 180,E1 -4870.517,E2 -4870.517} C_VEL
LIN {X 0,Y 524.744,Z 696.267,A -85,B 0,C 180,E1 -4870.832,E2 -4870.832} C_VEL
LIN {X 0,Y 524.927,Z 642.633,A -85,B 0,C 180,E1 -4871.585,E2 -4871.585} C_VEL
LIN {X 0,Y 524.83,Z 622.8,A -85,B 0,C 180,E1 -4871.86,E2 -4871.86} C_VEL
LIN {X 0,Y 524.086,Z 616.382,A -85,B 0,C 180,E1 -4871.995,E2 -4871.995} C_VEL
LIN {X 0,Y 524.461,Z 594.376,A -85,B 0,C 180,E1 -4875.098,E2 -4875.098} C_VEL
LIN {X 0,Y 524.903,Z 570.422,A -85,B 0,C 180,E1 -4878.521,E2 -4878.521} C_VEL
LIN {X 0,Y 525.322,Z 550.389,A -85,B 0,C 180,E1 -4881.381,E2 -4881.381} C_VEL
LIN {X 0,Y 525.727,Z 531.696,A -85,B 0,C 180,E1 -4884.062,E2 -4884.062} C_VEL
LIN {X 0,Y 525.487,Z 526.89,A -85,B 0,C 180,E1 -4884.763,E2 -4884.763} C_VEL
LIN {X 0,Y 524.006,Z 519.317,A -85,B 0,C 180,E1 -4885.957,E2 -4885.957} C_VEL
LIN {X 0,Y 523.943,Z 519.219,A -85,B 0,C 180,E1 -4888.875,E2 -4888.875} C_VEL
LIN {X 0,Y 523.938,Z 519.219,A -85,B 0,C 180,E1 -4890.265,E2 -4890.265} C_VEL
LIN {X 0,Y 523.282,Z 519.3,A -85,B 0,C 180,E1 -4890.907,E2 -4890.907} C_VEL
LIN {X 0,Y 520.411,Z 519.662,A -85,B 0,C 180,E1 -4891.949,E2 -4891.949} C_VEL
LIN {X 0,Y 517.989,Z 519.96,A -85,B 0,C 180,E1 -4892.788,E2 -4892.788} C_VEL
LIN {X 0,Y 516.97,Z 520.091,A -85,B 0,C 180,E1 -4893.436,E2 -4893.436} C_VEL
LIN {X 0,Y 516.898,Z 520.097,A -85,B 0,C 180,E1 -4893.656,E2 -4893.656} C_VEL
LIN {X 0,Y 516.882,Z 520.096,A -85,B 0,C 180,E1 -4896.746,E2 -4896.746} C_VEL
LIN {X 0,Y 516.886,Z 520.094,A -85,B 0,C 180,E1 -4899.721,E2 -4899.721} C_VEL
LIN {X 0,Y 516.915,Z 520.08,A -85,B 0,C 180,E1 -4901.775,E2 -4901.775} C_VEL
LIN {X 0,Y 516.899,Z 520.093,A -85,B 0,C 180,E1 -4905.007,E2 -4905.007} C_VEL
LIN {X 0,Y 516.918,Z 520.089,A -85,B 0,C 180,E1 -4908.399,E2 -4908.399} C_VEL
LIN {X 0,Y 516.883,Z 520.095,A -85,B 0,C 180,E1 -4911.284,E2 -4911.284} C_VEL
LIN {X 0,Y 516.875,Z 520.096,A -85,B 0,C 180,E1 -4914.219,E2 -4914.219} C_VEL
LIN {X 0,Y 516.885,Z 520.103,A -85,B 0,C 180,E1 -4917.052,E2 -4917.052} C_VEL
LIN {X 0,Y 516.897,Z 520.095,A -85,B 0,C 180,E1 -4919.796,E2 -4919.796} C_VEL
LIN {X 0,Y 516.931,Z 520.093,A -85,B 0,C 180,E1 -4922.467,E2 -4922.467} C_VEL
LIN {X 0,Y 516.908,Z 520.094,A -85,B 0,C 180,E1 -4925.071,E2 -4925.071} C_VEL
LIN {X 0,Y 516.893,Z 520.097,A -85,B 0,C 180,E1 -4928.462,E2 -4928.462} C_VEL
LIN {X 0,Y 516.973,Z 520.261,A -85,B 0,C 180,E1 -4929.248,E2 -4929.248} C_VEL
LIN {X 0,Y 517.793,Z 525.613,A -85,B 0,C 180,E1 -4930.37,E2 -4930.37} C_VEL
LIN {X 0,Y 517.387,Z 541.23,A -85,B 0,C 180,E1 -4933.425,E2 -4933.425} C_VEL
LIN {X 0,Y 517.249,Z 547.885,A -85,B 0,C 180,E1 -4934.662,E2 -4934.662} C_VEL
LIN {X 0,Y 518.104,Z 552.977,A -85,B 0,C 180,E1 -4934.794,E2 -4934.794} C_VEL
LIN {X 0,Y 519.106,Z 559.438,A -85,B 0,C 180,E1 -4934.916,E2 -4934.916} C_VEL
LIN {X 0,Y 518.652,Z 654.655,A -85,B 0,C 180,E1 -4936.257,E2 -4936.257} C_VEL
LIN {X 0,Y 518.469,Z 667.843,A -85,B 0,C 180,E1 -4936.602,E2 -4936.602} C_VEL
LIN {X 0,Y 518.205,Z 679.939,A -85,B 0,C 180,E1 -4937.069,E2 -4937.069} C_VEL
LIN {X 0,Y 517.96,Z 691.547,A -85,B 0,C 180,E1 -4937.673,E2 -4937.673} C_VEL
LIN {X 0,Y 517.639,Z 703.016,A -85,B 0,C 180,E1 -4938.447,E2 -4938.447} C_VEL
LIN {X 0,Y 517.306,Z 713.494,A -85,B 0,C 180,E1 -4939.332,E2 -4939.332} C_VEL
LIN {X 0,Y 517.055,Z 722.051,A -85,B 0,C 180,E1 -4940.217,E2 -4940.217} C_VEL
LIN {X 0,Y 516.835,Z 729.933,A -85,B 0,C 180,E1 -4941.2,E2 -4941.2} C_VEL
LIN {X 0,Y 516.602,Z 737.639,A -85,B 0,C 180,E1 -4942.377,E2 -4942.377} C_VEL
LIN {X 0,Y 516.45,Z 744.708,A -85,B 0,C 180,E1 -4943.749,E2 -4943.749} C_VEL
LIN {X 0,Y 516.314,Z 749.42,A -85,B 0,C 180,E1 -4944.923,E2 -4944.923} C_VEL
LIN {X 0,Y 516.373,Z 753.023,A -85,B 0,C 180,E1 -4946.097,E2 -4946.097} C_VEL
LIN {X 0,Y 516.283,Z 754.889,A -85,B 0,C 180,E1 -4946.878,E2 -4946.878} C_VEL
LIN {X 0,Y 516.261,Z 756.298,A -85,B 0,C 180,E1 -4947.659,E2 -4947.659} C_VEL
LIN {X 0,Y 516.16,Z 757.917,A -85,B 0,C 180,E1 -4949.219,E2 -4949.219} C_VEL
LIN {X 0,Y 516.155,Z 758.155,A -85,B 0,C 180,E1 -4949.999,E2 -4949.999} C_VEL
LIN {X 0,Y 516.16,Z 757.973,A -85,B 0,C 180,E1 -4950.779,E2 -4950.779} C_VEL
LIN {X 0,Y 516.261,Z 756.429,A -85,B 0,C 180,E1 -4952.34,E2 -4952.34} C_VEL
LIN {X 0,Y 516.283,Z 755.076,A -85,B 0,C 180,E1 -4953.121,E2 -4953.121} C_VEL
LIN {X 0,Y 516.361,Z 752.212,A -85,B 0,C 180,E1 -4954.292,E2 -4954.292} C_VEL
LIN {X 0,Y 516.403,Z 748.332,A -85,B 0,C 180,E1 -4955.466,E2 -4955.466} C_VEL
LIN {X 0,Y 516.481,Z 742.515,A -85,B 0,C 180,E1 -4956.808,E2 -4956.808} C_VEL
LIN {X 0,Y 516.653,Z 735.808,A -85,B 0,C 180,E1 -4958.014,E2 -4958.014} C_VEL
LIN {X 0,Y 516.88,Z 727.661,A -85,B 0,C 180,E1 -4959.192,E2 -4959.192} C_VEL
LIN {X 0,Y 517.098,Z 719.324,A -85,B 0,C 180,E1 -4960.176,E2 -4960.176} C_VEL
LIN {X 0,Y 517.475,Z 709.029,A -85,B 0,C 180,E1 -4961.158,E2 -4961.158} C_VEL
LIN {X 0,Y 517.789,Z 697.501,A -85,B 0,C 180,E1 -4962.038,E2 -4962.038} C_VEL
LIN {X 0,Y 518.082,Z 685.861,A -85,B 0,C 180,E1 -4962.734,E2 -4962.734} C_VEL
LIN {X 0,Y 518.365,Z 673.841,A -85,B 0,C 180,E1 -4963.275,E2 -4963.275} C_VEL
LIN {X 0,Y 518.592,Z 660.779,A -85,B 0,C 180,E1 -4963.693,E2 -4963.693} C_VEL
LIN {X 0,Y 518.751,Z 648.311,A -85,B 0,C 180,E1 -4963.939,E2 -4963.939} C_VEL
LIN {X 0,Y 519.055,Z 558.166,A -85,B 0,C 180,E1 -4965.194,E2 -4965.194} C_VEL
LIN {X 0,Y 517.294,Z 548.215,A -85,B 0,C 180,E1 -4965.406,E2 -4965.406} C_VEL
LIN {X 0,Y 517.24,Z 547.422,A -85,B 0,C 180,E1 -4965.485,E2 -4965.485} C_VEL
LIN {X 0,Y 517.619,Z 532.327,A -85,B 0,C 180,E1 -4968.401,E2 -4968.401} C_VEL
LIN {X 0,Y 517.715,Z 525.036,A -85,B 0,C 180,E1 -4969.838,E2 -4969.838} C_VEL
LIN {X 0,Y 516.926,Z 520.124,A -85,B 0,C 180,E1 -4970.908,E2 -4970.908} C_VEL
LIN {X 0,Y 516.904,Z 520.094,A -85,B 0,C 180,E1 -4974.362,E2 -4974.362} C_VEL
LIN {X 0,Y 516.926,Z 520.089,A -85,B 0,C 180,E1 -4976.657,E2 -4976.657} C_VEL
LIN {X 0,Y 516.911,Z 520.094,A -85,B 0,C 180,E1 -4979.523,E2 -4979.523} C_VEL
LIN {X 0,Y 516.9,Z 520.093,A -85,B 0,C 180,E1 -4982.543,E2 -4982.543} C_VEL
LIN {X 0,Y 516.881,Z 520.103,A -85,B 0,C 180,E1 -4985.331,E2 -4985.331} C_VEL
LIN {X 0,Y 516.88,Z 520.098,A -85,B 0,C 180,E1 -4987.942,E2 -4987.942} C_VEL
LIN {X 0,Y 516.883,Z 520.094,A -85,B 0,C 180,E1 -4990.74,E2 -4990.74} C_VEL
LIN {X 0,Y 516.902,Z 520.094,A -85,B 0,C 180,E1 -4992.828,E2 -4992.828} C_VEL
LIN {X 0,Y 516.919,Z 520.09,A -85,B 0,C 180,E1 -4995.009,E2 -4995.009} C_VEL
LIN {X 0,Y 516.918,Z 520.09,A -85,B 0,C 180,E1 -4998.397,E2 -4998.397} C_VEL
LIN {X 0,Y 516.902,Z 520.093,A -85,B 0,C 180,E1 -5001.286,E2 -5001.286} C_VEL
LIN {X 0,Y 516.887,Z 520.095,A -85,B 0,C 180,E1 -5004.221,E2 -5004.221} C_VEL
LIN {X 0,Y 516.893,Z 520.096,A -85,B 0,C 180,E1 -5007.053,E2 -5007.053} C_VEL
LIN {X 0,Y 516.896,Z 520.098,A -85,B 0,C 180,E1 -5009.796,E2 -5009.796} C_VEL
LIN {X 0,Y 516.924,Z 520.086,A -85,B 0,C 180,E1 -5012.467,E2 -5012.467} C_VEL
LIN {X 0,Y 516.906,Z 520.095,A -85,B 0,C 180,E1 -5015.071,E2 -5015.071} C_VEL
LIN {X 0,Y 516.88,Z 520.092,A -85,B 0,C 180,E1 -5018.462,E2 -5018.462} C_VEL
LIN {X 0,Y 516.898,Z 520.094,A -85,B 0,C 180,E1 -5020.955,E2 -5020.955} C_VEL
LIN {X 0,Y 516.911,Z 520.096,A -85,B 0,C 180,E1 -5023.41,E2 -5023.41} C_VEL
LIN {X 0,Y 516.888,Z 520.098,A -85,B 0,C 180,E1 -5025.833,E2 -5025.833} C_VEL
LIN {X 0,Y 516.957,Z 520.085,A -85,B 0,C 180,E1 -5028.233,E2 -5028.233} C_VEL
LIN {X 0,Y 516.965,Z 520.088,A -85,B 0,C 180,E1 -5031.4,E2 -5031.4} C_VEL
LIN {X 0,Y 517.003,Z 520.085,A -85,B 0,C 180,E1 -5033.757,E2 -5033.757} C_VEL
LIN {X 0,Y 517.077,Z 520.076,A -85,B 0,C 180,E1 -5037.663,E2 -5037.663} C_VEL
LIN {X 0,Y 517.088,Z 520.07,A -85,B 0,C 180,E1 -5040.779,E2 -5040.779} C_VEL
LIN {X 0,Y 517.009,Z 520.08,A -85,B 0,C 180,E1 -5043.117,E2 -5043.117} C_VEL
LIN {X 0,Y 517.003,Z 520.081,A -85,B 0,C 180,E1 -5046.243,E2 -5046.243} C_VEL
LIN {X 0,Y 516.947,Z 520.092,A -85,B 0,C 180,E1 -5049.389,E2 -5049.389} C_VEL
LIN {X 0,Y 516.976,Z 520.089,A -85,B 0,C 180,E1 -5051.824,E2 -5051.824} C_VEL
LIN {X 0,Y 516.936,Z 520.09,A -85,B 0,C 180,E1 -5055.147,E2 -5055.147} C_VEL
LIN {X 0,Y 516.919,Z 520.092,A -85,B 0,C 180,E1 -5058.222,E2 -5058.222} C_VEL
LIN {X 0,Y 516.906,Z 520.091,A -85,B 0,C 180,E1 -5060.702,E2 -5060.702} C_VEL
LIN {X 0,Y 516.904,Z 520.095,A -85,B 0,C 180,E1 -5064.072,E2 -5064.072} C_VEL
LIN {X 0,Y 516.923,Z 520.087,A -85,B 0,C 180,E1 -5066.658,E2 -5066.658} C_VEL
LIN {X 0,Y 516.905,Z 520.1,A -85,B 0,C 180,E1 -5069.525,E2 -5069.525} C_VEL
LIN {X 0,Y 516.895,Z 520.093,A -85,B 0,C 180,E1 -5072.545,E2 -5072.545} C_VEL
LIN {X 0,Y 516.879,Z 520.098,A -85,B 0,C 180,E1 -5075.333,E2 -5075.333} C_VEL
LIN {X 0,Y 516.876,Z 520.1,A -85,B 0,C 180,E1 -5077.944,E2 -5077.944} C_VEL
LIN {X 0,Y 516.881,Z 520.095,A -85,B 0,C 180,E1 -5080.742,E2 -5080.742} C_VEL
LIN {X 0,Y 516.879,Z 520.091,A -85,B 0,C 180,E1 -5082.832,E2 -5082.832} C_VEL
LIN {X 0,Y 516.918,Z 520.092,A -85,B 0,C 180,E1 -5085.011,E2 -5085.011} C_VEL
LIN {X 0,Y 516.92,Z 520.092,A -85,B 0,C 180,E1 -5088.398,E2 -5088.398} C_VEL
LIN {X 0,Y 516.884,Z 520.096,A -85,B 0,C 180,E1 -5091.286,E2 -5091.286} C_VEL
LIN {X 0,Y 516.885,Z 520.098,A -85,B 0,C 180,E1 -5094.222,E2 -5094.222} C_VEL
LIN {X 0,Y 516.896,Z 520.09,A -85,B 0,C 180,E1 -5097.054,E2 -5097.054} C_VEL
LIN {X 0,Y 516.891,Z 520.079,A -85,B 0,C 180,E1 -5099.797,E2 -5099.797} C_VEL
LIN {X 0,Y 516.928,Z 520.089,A -85,B 0,C 180,E1 -5102.468,E2 -5102.468} C_VEL
LIN {X 0,Y 516.922,Z 520.118,A -85,B 0,C 180,E1 -5105.518,E2 -5105.518} C_VEL
LIN {X 0,Y 516.937,Z 520.334,A -85,B 0,C 180,E1 -5105.63,E2 -5105.63} C_VEL
LIN {X 0,Y 518.489,Z 529.102,A -85,B 0,C 180,E1 -5107.18,E2 -5107.18} C_VEL
LIN {X 0,Y 518.038,Z 546.242,A -85,B 0,C 180,E1 -5109.973,E2 -5109.973} C_VEL
LIN {X 0,Y 517.566,Z 564,A -85,B 0,C 180,E1 -5112.823,E2 -5112.823} C_VEL
LIN {X 0,Y 517.372,Z 575.517,A -85,B 0,C 180,E1 -5114.617,E2 -5114.617} C_VEL
LIN {X 0,Y 519.137,Z 588.028,A -85,B 0,C 180,E1 -5114.867,E2 -5114.867} C_VEL
LIN {X 0,Y 518.661,Z 683.537,A -85,B 0,C 180,E1 -5116.209,E2 -5116.209} C_VEL
LIN {X 0,Y 518.409,Z 696.802,A -85,B 0,C 180,E1 -5116.551,E2 -5116.551} C_VEL
LIN {X 0,Y 518.112,Z 710.093,A -85,B 0,C 180,E1 -5117.067,E2 -5117.067} C_VEL
LIN {X 0,Y 517.846,Z 722.403,A -85,B 0,C 180,E1 -5117.73,E2 -5117.73} C_VEL
LIN {X 0,Y 517.527,Z 734.155,A -85,B 0,C 180,E1 -5118.545,E2 -5118.545} C_VEL
LIN {X 0,Y 517.239,Z 744.351,A -85,B 0,C 180,E1 -5119.431,E2 -5119.431} C_VEL
LIN {X 0,Y 516.951,Z 753.528,A -85,B 0,C 180,E1 -5120.414,E2 -5120.414} C_VEL
LIN {X 0,Y 516.699,Z 762.469,A -85,B 0,C 180,E1 -5121.593,E2 -5121.593} C_VEL
LIN {X 0,Y 516.509,Z 769.667,A -85,B 0,C 180,E1 -5122.77,E2 -5122.77} C_VEL
LIN {X 0,Y 516.453,Z 776.221,A -85,B 0,C 180,E1 -5124.143,E2 -5124.143} C_VEL
LIN {X 0,Y 516.271,Z 780.555,A -85,B 0,C 180,E1 -5125.316,E2 -5125.316} C_VEL
LIN {X 0,Y 516.354,Z 782.857,A -85,B 0,C 180,E1 -5126.098,E2 -5126.098} C_VEL
LIN {X 0,Y 516.282,Z 784.716,A -85,B 0,C 180,E1 -5126.879,E2 -5126.879} C_VEL
LIN {X 0,Y 516.26,Z 786.11,A -85,B 0,C 180,E1 -5127.66,E2 -5127.66} C_VEL
LIN {X 0,Y 516.16,Z 787.708,A -85,B 0,C 180,E1 -5129.221,E2 -5129.221} C_VEL
LIN {X 0,Y 516.154,Z 787.924,A -85,B 0,C 180,E1 -5130.001,E2 -5130.001} C_VEL
LIN {X 0,Y 516.192,Z 787.1,A -85,B 0,C 180,E1 -5131.561,E2 -5131.561} C_VEL
LIN {X 0,Y 516.26,Z 786.105,A -85,B 0,C 180,E1 -5132.341,E2 -5132.341} C_VEL
LIN {X 0,Y 516.283,Z 784.71,A -85,B 0,C 180,E1 -5133.122,E2 -5133.122} C_VEL
LIN {X 0,Y 516.327,Z 781.779,A -85,B 0,C 180,E1 -5134.294,E2 -5134.294} C_VEL
LIN {X 0,Y 516.405,Z 777.81,A -85,B 0,C 180,E1 -5135.467,E2 -5135.467} C_VEL
LIN {X 0,Y 516.465,Z 772.519,A -85,B 0,C 180,E1 -5136.679,E2 -5136.679} C_VEL
LIN {X 0,Y 516.598,Z 766.257,A -85,B 0,C 180,E1 -5137.82,E2 -5137.82} C_VEL
LIN {X 0,Y 516.811,Z 758.229,A -85,B 0,C 180,E1 -5138.998,E2 -5138.998} C_VEL
LIN {X 0,Y 517.053,Z 750.048,A -85,B 0,C 180,E1 -5139.981,E2 -5139.981} C_VEL
LIN {X 0,Y 517.334,Z 740.072,A -85,B 0,C 180,E1 -5140.964,E2 -5140.964} C_VEL
LIN {X 0,Y 517.635,Z 730.23,A -85,B 0,C 180,E1 -5141.751,E2 -5141.751} C_VEL
LIN {X 0,Y 517.923,Z 719.06,A -85,B 0,C 180,E1 -5142.468,E2 -5142.468} C_VEL
LIN {X 0,Y 518.189,Z 706.684,A -85,B 0,C 180,E1 -5143.081,E2 -5143.081} C_VEL
LIN {X 0,Y 518.474,Z 693.641,A -85,B 0,C 180,E1 -5143.548,E2 -5143.548} C_VEL
LIN {X 0,Y 518.695,Z 680.623,A -85,B 0,C 180,E1 -5143.842,E2 -5143.842} C_VEL
LIN {X 0,Y 518.985,Z 585.984,A -85,B 0,C 180,E1 -5145.166,E2 -5145.166} C_VEL
LIN {X 0,Y 517.347,Z 575.434,A -85,B 0,C 180,E1 -5145.389,E2 -5145.389} C_VEL
LIN {X 0,Y 517.816,Z 555.094,A -85,B 0,C 180,E1 -5148.6,E2 -5148.6} C_VEL
LIN {X 0,Y 518.288,Z 536.033,A -85,B 0,C 180,E1 -5151.686,E2 -5151.686} C_VEL
LIN {X 0,Y 518.525,Z 529.043,A -85,B 0,C 180,E1 -5152.829,E2 -5152.829} C_VEL
LIN {X 0,Y 516.959,Z 520.311,A -85,B 0,C 180,E1 -5154.376,E2 -5154.376} C_VEL
LIN {X 0,Y 516.93,Z 520.096,A -85,B 0,C 180,E1 -5156.658,E2 -5156.658} C_VEL
LIN {X 0,Y 516.915,Z 520.086,A -85,B 0,C 180,E1 -5159.524,E2 -5159.524} C_VEL
LIN {X 0,Y 516.9,Z 520.098,A -85,B 0,C 180,E1 -5162.544,E2 -5162.544} C_VEL
LIN {X 0,Y 516.87,Z 520.097,A -85,B 0,C 180,E1 -5165.33,E2 -5165.33} C_VEL
LIN {X 0,Y 516.884,Z 520.1,A -85,B 0,C 180,E1 -5167.943,E2 -5167.943} C_VEL
LIN {X 0,Y 516.887,Z 520.098,A -85,B 0,C 180,E1 -5170.742,E2 -5170.742} C_VEL
LIN {X 0,Y 516.888,Z 520.097,A -85,B 0,C 180,E1 -5172.831,E2 -5172.831} C_VEL
LIN {X 0,Y 516.898,Z 520.095,A -85,B 0,C 180,E1 -5175.007,E2 -5175.007} C_VEL
LIN {X 0,Y 516.916,Z 520.098,A -85,B 0,C 180,E1 -5178.399,E2 -5178.399} C_VEL
LIN {X 0,Y 516.884,Z 520.096,A -85,B 0,C 180,E1 -5181.284,E2 -5181.284} C_VEL
LIN {X 0,Y 516.891,Z 520.103,A -85,B 0,C 180,E1 -5184.221,E2 -5184.221} C_VEL
LIN {X 0,Y 516.898,Z 520.095,A -85,B 0,C 180,E1 -5187.053,E2 -5187.053} C_VEL
LIN {X 0,Y 516.895,Z 520.1,A -85,B 0,C 180,E1 -5189.796,E2 -5189.796} C_VEL
LIN {X 0,Y 516.932,Z 520.097,A -85,B 0,C 180,E1 -5192.468,E2 -5192.468} C_VEL
LIN {X 0,Y 516.966,Z 520.223,A -85,B 0,C 180,E1 -5194.429,E2 -5194.429} C_VEL
LIN {X 0,Y 518.445,Z 528.477,A -85,B 0,C 180,E1 -5195.63,E2 -5195.63} C_VEL
LIN {X 0,Y 518.202,Z 547.987,A -85,B 0,C 180,E1 -5198.311,E2 -5198.311} C_VEL
LIN {X 0,Y 517.915,Z 565.795,A -85,B 0,C 180,E1 -5200.788,E2 -5200.788} C_VEL
LIN {X 0,Y 517.633,Z 583.331,A -85,B 0,C 180,E1 -5203.231,E2 -5203.231} C_VEL
LIN {X 0,Y 517.225,Z 602.682,A -85,B 0,C 180,E1 -5206.043,E2 -5206.043} C_VEL
LIN {X 0,Y 517.103,Z 616.458,A -85,B 0,C 180,E1 -5207.937,E2 -5207.937} C_VEL
LIN {X 0,Y 517.988,Z 625.749,A -85,B 0,C 180,E1 -5208.121,E2 -5208.121} C_VEL
LIN {X 0,Y 517.779,Z 695.772,A -85,B 0,C 180,E1 -5209.12,E2 -5209.12} C_VEL
LIN {X 0,Y 517.638,Z 706.763,A -85,B 0,C 180,E1 -5209.414,E2 -5209.414} C_VEL
LIN {X 0,Y 517.436,Z 717.2,A -85,B 0,C 180,E1 -5209.83,E2 -5209.83} C_VEL
LIN {X 0,Y 517.233,Z 727.825,A -85,B 0,C 180,E1 -5210.419,E2 -5210.419} C_VEL
LIN {X 0,Y 517.027,Z 737.276,A -85,B 0,C 180,E1 -5211.105,E2 -5211.105} C_VEL
LIN {X 0,Y 516.856,Z 744.874,A -85,B 0,C 180,E1 -5211.792,E2 -5211.792} C_VEL
LIN {X 0,Y 516.66,Z 753.565,A -85,B 0,C 180,E1 -5212.772,E2 -5212.772} C_VEL
LIN {X 0,Y 516.595,Z 760.383,A -85,B 0,C 180,E1 -5213.752,E2 -5213.752} C_VEL
LIN {X 0,Y 516.355,Z 766.736,A -85,B 0,C 180,E1 -5214.924,E2 -5214.924} C_VEL
LIN {X 0,Y 516.387,Z 771.486,A -85,B 0,C 180,E1 -5216.098,E2 -5216.098} C_VEL
LIN {X 0,Y 516.296,Z 773.851,A -85,B 0,C 180,E1 -5216.879,E2 -5216.879} C_VEL
LIN {X 0,Y 516.262,Z 775.651,A -85,B 0,C 180,E1 -5217.659,E2 -5217.659} C_VEL
LIN {X 0,Y 516.19,Z 776.944,A -85,B 0,C 180,E1 -5218.44,E2 -5218.44} C_VEL
LIN {X 0,Y 516.157,Z 777.738,A -85,B 0,C 180,E1 -5219.22,E2 -5219.22} C_VEL
LIN {X 0,Y 516.152,Z 778.029,A -85,B 0,C 180,E1 -5220,E2 -5220} C_VEL
LIN {X 0,Y 516.159,Z 777.807,A -85,B 0,C 180,E1 -5220.78,E2 -5220.78} C_VEL
LIN {X 0,Y 516.192,Z 777.068,A -85,B 0,C 180,E1 -5221.56,E2 -5221.56} C_VEL
LIN {X 0,Y 516.263,Z 775.827,A -85,B 0,C 180,E1 -5222.341,E2 -5222.341} C_VEL
LIN {X 0,Y 516.327,Z 773.001,A -85,B 0,C 180,E1 -5223.512,E2 -5223.512} C_VEL
LIN {X 0,Y 516.314,Z 768.865,A -85,B 0,C 180,E1 -5224.685,E2 -5224.685} C_VEL
LIN {X 0,Y 516.532,Z 763.2,A -85,B 0,C 180,E1 -5225.857,E2 -5225.857} C_VEL
LIN {X 0,Y 516.596,Z 756.888,A -85,B 0,C 180,E1 -5226.868,E2 -5226.868} C_VEL
LIN {X 0,Y 516.739,Z 749.43,A -85,B 0,C 180,E1 -5227.817,E2 -5227.817} C_VEL
LIN {X 0,Y 516.971,Z 740.679,A -85,B 0,C 180,E1 -5228.699,E2 -5228.699} C_VEL
LIN {X 0,Y 517.2,Z 730.691,A -85,B 0,C 180,E1 -5229.483,E2 -5229.483} C_VEL
LIN {X 0,Y 517.398,Z 721.028,A -85,B 0,C 180,E1 -5230.072,E2 -5230.072} C_VEL
LIN {X 0,Y 517.57,Z 709.465,A -85,B 0,C 180,E1 -5230.588,E2 -5230.588} C_VEL
LIN {X 0,Y 517.699,Z 697.886,A -85,B 0,C 180,E1 -5230.931,E2 -5230.931} C_VEL
LIN {X 0,Y 517.885,Z 677.687,A -85,B 0,C 180,E1 -5231.249,E2 -5231.249} C_VEL
LIN {X 0,Y 517.896,Z 623.504,A -85,B 0,C 180,E1 -5232.007,E2 -5232.007} C_VEL
LIN {X 0,Y 517.067,Z 616.379,A -85,B 0,C 180,E1 -5232.158,E2 -5232.158} C_VEL
LIN {X 0,Y 517.447,Z 595.007,A -85,B 0,C 180,E1 -5235.207,E2 -5235.207} C_VEL
LIN {X 0,Y 517.912,Z 571.711,A -85,B 0,C 180,E1 -5238.555,E2 -5238.555} C_VEL
LIN {X 0,Y 518.37,Z 551.466,A -85,B 0,C 180,E1 -5241.473,E2 -5241.473} C_VEL
LIN {X 0,Y 518.782,Z 532.66,A -85,B 0,C 180,E1 -5244.192,E2 -5244.192} C_VEL
LIN {X 0,Y 518.545,Z 528.244,A -85,B 0,C 180,E1 -5244.844,E2 -5244.844} C_VEL
LIN {X 0,Y 516.972,Z 520.177,A -85,B 0,C 180,E1 -5246.134,E2 -5246.134} C_VEL
LIN {X 0,Y 516.925,Z 520.096,A -85,B 0,C 180,E1 -5249.304,E2 -5249.304} C_VEL
LIN {X 0,Y 516.899,Z 520.094,A -85,B 0,C 180,E1 -5252.543,E2 -5252.543} C_VEL
LIN {X 0,Y 516.898,Z 520.097,A -85,B 0,C 180,E1 -5253.656,E2 -5253.656} C_VEL
LIN {X 0,Y 516.259,Z 520.181,A -85,B 0,C 180,E1 -5254.306,E2 -5254.306} C_VEL
LIN {X 0,Y 513.395,Z 520.536,A -85,B 0,C 180,E1 -5255.361,E2 -5255.361} C_VEL
LIN {X 0,Y 510.954,Z 520.836,A -85,B 0,C 180,E1 -5256.211,E2 -5256.211} C_VEL
LIN {X 0,Y 509.904,Z 520.966,A -85,B 0,C 180,E1 -5256.868,E2 -5256.868} C_VEL
LIN {X 0,Y 509.819,Z 520.978,A -85,B 0,C 180,E1 -5257.09,E2 -5257.09} C_VEL
LIN {X 0,Y 509.838,Z 520.976,A -85,B 0,C 180,E1 -5259.47,E2 -5259.47} C_VEL
LIN {X 0,Y 509.823,Z 520.958,A -85,B 0,C 180,E1 -5262.491,E2 -5262.491} C_VEL
LIN {X 0,Y 509.843,Z 520.977,A -85,B 0,C 180,E1 -5265.33,E2 -5265.33} C_VEL
LIN {X 0,Y 509.86,Z 520.969,A -85,B 0,C 180,E1 -5268.574,E2 -5268.574} C_VEL
LIN {X 0,Y 509.855,Z 520.971,A -85,B 0,C 180,E1 -5271.786,E2 -5271.786} C_VEL
LIN {X 0,Y 509.834,Z 520.976,A -85,B 0,C 180,E1 -5274.622,E2 -5274.622} C_VEL
LIN {X 0,Y 509.864,Z 520.973,A -85,B 0,C 180,E1 -5277.481,E2 -5277.481} C_VEL
LIN {X 0,Y 509.863,Z 520.972,A -85,B 0,C 180,E1 -5280.273,E2 -5280.273} C_VEL
LIN {X 0,Y 509.889,Z 520.974,A -85,B 0,C 180,E1 -5282.944,E2 -5282.944} C_VEL
LIN {X 0,Y 509.86,Z 520.968,A -85,B 0,C 180,E1 -5285.573,E2 -5285.573} C_VEL
LIN {X 0,Y 509.934,Z 521.09,A -85,B 0,C 180,E1 -5289.076,E2 -5289.076} C_VEL
LIN {X 0,Y 510.819,Z 526.819,A -85,B 0,C 180,E1 -5290.3,E2 -5290.3} C_VEL
LIN {X 0,Y 510.406,Z 542.458,A -85,B 0,C 180,E1 -5293.398,E2 -5293.398} C_VEL
LIN {X 0,Y 510.272,Z 548.115,A -85,B 0,C 180,E1 -5294.452,E2 -5294.452} C_VEL
LIN {X 0,Y 511.943,Z 557.381,A -85,B 0,C 180,E1 -5294.667,E2 -5294.667} C_VEL
LIN {X 0,Y 512.247,Z 561.174,A -85,B 0,C 180,E1 -5294.73,E2 -5294.73} C_VEL
LIN {X 0,Y 511.778,Z 654.888,A -85,B 0,C 180,E1 -5296.069,E2 -5296.069} C_VEL
LIN {X 0,Y 511.568,Z 668.066,A -85,B 0,C 180,E1 -5296.417,E2 -5296.417} C_VEL
LIN {X 0,Y 511.3,Z 680.157,A -85,B 0,C 180,E1 -5296.891,E2 -5296.891} C_VEL
LIN {X 0,Y 511.012,Z 691.806,A -85,B 0,C 180,E1 -5297.505,E2 -5297.505} C_VEL
LIN {X 0,Y 510.69,Z 703.227,A -85,B 0,C 180,E1 -5298.288,E2 -5298.288} C_VEL
LIN {X 0,Y 510.326,Z 713.705,A -85,B 0,C 180,E1 -5299.184,E2 -5299.184} C_VEL
LIN {X 0,Y 510.058,Z 722.261,A -85,B 0,C 180,E1 -5300.082,E2 -5300.082} C_VEL
LIN {X 0,Y 509.821,Z 730.142,A -85,B 0,C 180,E1 -5301.078,E2 -5301.078} C_VEL
LIN {X 0,Y 509.56,Z 737.848,A -85,B 0,C 180,E1 -5302.271,E2 -5302.271} C_VEL
LIN {X 0,Y 509.388,Z 744.915,A -85,B 0,C 180,E1 -5303.662,E2 -5303.662} C_VEL
LIN {X 0,Y 509.248,Z 749.627,A -85,B 0,C 180,E1 -5304.853,E2 -5304.853} C_VEL
LIN {X 0,Y 509.303,Z 753.227,A -85,B 0,C 180,E1 -5306.043,E2 -5306.043} C_VEL
LIN {X 0,Y 509.202,Z 755.093,A -85,B 0,C 180,E1 -5306.835,E2 -5306.835} C_VEL
LIN {X 0,Y 509.19,Z 756.501,A -85,B 0,C 180,E1 -5307.626,E2 -5307.626} C_VEL
LIN {X 0,Y 509.074,Z 758.122,A -85,B 0,C 180,E1 -5309.208,E2 -5309.208} C_VEL
LIN {X 0,Y 509.066,Z 758.36,A -85,B 0,C 180,E1 -5309.999,E2 -5309.999} C_VEL
LIN {X 0,Y 509.073,Z 758.177,A -85,B 0,C 180,E1 -5310.79,E2 -5310.79} C_VEL
LIN {X 0,Y 509.19,Z 756.632,A -85,B 0,C 180,E1 -5312.372,E2 -5312.372} C_VEL
LIN {X 0,Y 509.202,Z 755.28,A -85,B 0,C 180,E1 -5313.164,E2 -5313.164} C_VEL
LIN {X 0,Y 509.282,Z 752.416,A -85,B 0,C 180,E1 -5314.352,E2 -5314.352} C_VEL
LIN {X 0,Y 509.345,Z 748.534,A -85,B 0,C 180,E1 -5315.542,E2 -5315.542} C_VEL
LIN {X 0,Y 509.41,Z 743.532,A -85,B 0,C 180,E1 -5316.733,E2 -5316.733} C_VEL
LIN {X 0,Y 509.595,Z 737.231,A -85,B 0,C 180,E1 -5317.926,E2 -5317.926} C_VEL
LIN {X 0,Y 509.802,Z 729.34,A -85,B 0,C 180,E1 -5319.121,E2 -5319.121} C_VEL
LIN {X 0,Y 510.103,Z 719.523,A -85,B 0,C 180,E1 -5320.317,E2 -5320.317} C_VEL
LIN {X 0,Y 510.509,Z 709.225,A -85,B 0,C 180,E1 -5321.313,E2 -5321.313} C_VEL
LIN {X 0,Y 510.834,Z 698.335,A -85,B 0,C 180,E1 -5322.159,E2 -5322.159} C_VEL
LIN {X 0,Y 511.09,Z 687.868,A -85,B 0,C 180,E1 -5322.81,E2 -5322.81} C_VEL
LIN {X 0,Y 511.428,Z 676.549,A -85,B 0,C 180,E1 -5323.357,E2 -5323.357} C_VEL
LIN {X 0,Y 511.651,Z 663.702,A -85,B 0,C 180,E1 -5323.807,E2 -5323.807} C_VEL
LIN {X 0,Y 511.865,Z 650.025,A -85,B 0,C 180,E1 -5324.105,E2 -5324.105} C_VEL
LIN {X 0,Y 512.139,Z 558.593,A -85,B 0,C 180,E1 -5325.4,E2 -5325.4} C_VEL
LIN {X 0,Y 510.31,Z 548.445,A -85,B 0,C 180,E1 -5325.62,E2 -5325.62} C_VEL
LIN {X 0,Y 510.257,Z 546.953,A -85,B 0,C 180,E1 -5325.814,E2 -5325.814} C_VEL
LIN {X 0,Y 510.701,Z 531.439,A -85,B 0,C 180,E1 -5328.867,E2 -5328.867} C_VEL
LIN {X 0,Y 510.644,Z 525.198,A -85,B 0,C 180,E1 -5330.124,E2 -5330.124} C_VEL
LIN {X 0,Y 509.881,Z 520.997,A -85,B 0,C 180,E1 -5331.079,E2 -5331.079} C_VEL
LIN {X 0,Y 509.871,Z 520.971,A -85,B 0,C 180,E1 -5334.425,E2 -5334.425} C_VEL
LIN {X 0,Y 509.885,Z 520.97,A -85,B 0,C 180,E1 -5337.055,E2 -5337.055} C_VEL
LIN {X 0,Y 509.856,Z 520.973,A -85,B 0,C 180,E1 -5339.75,E2 -5339.75} C_VEL
LIN {X 0,Y 509.876,Z 520.969,A -85,B 0,C 180,E1 -5342.774,E2 -5342.774} C_VEL
LIN {X 0,Y 509.841,Z 520.977,A -85,B 0,C 180,E1 -5345.58,E2 -5345.58} C_VEL
LIN {X 0,Y 509.849,Z 520.971,A -85,B 0,C 180,E1 -5348.337,E2 -5348.337} C_VEL
LIN {X 0,Y 509.856,Z 520.978,A -85,B 0,C 180,E1 -5351.424,E2 -5351.424} C_VEL
LIN {X 0,Y 509.853,Z 520.967,A -85,B 0,C 180,E1 -5354.667,E2 -5354.667} C_VEL
LIN {X 0,Y 509.857,Z 520.971,A -85,B 0,C 180,E1 -5358.102,E2 -5358.102} C_VEL
LIN {X 0,Y 509.872,Z 520.964,A -85,B 0,C 180,E1 -5360.65,E2 -5360.65} C_VEL
LIN {X 0,Y 509.832,Z 520.98,A -85,B 0,C 180,E1 -5363.647,E2 -5363.647} C_VEL
LIN {X 0,Y 509.858,Z 520.969,A -85,B 0,C 180,E1 -5366.539,E2 -5366.539} C_VEL
LIN {X 0,Y 509.845,Z 520.978,A -85,B 0,C 180,E1 -5369.334,E2 -5369.334} C_VEL
LIN {X 0,Y 509.89,Z 520.964,A -85,B 0,C 180,E1 -5372.054,E2 -5372.054} C_VEL
LIN {X 0,Y 509.872,Z 520.968,A -85,B 0,C 180,E1 -5374.704,E2 -5374.704} C_VEL
LIN {X 0,Y 509.849,Z 520.976,A -85,B 0,C 180,E1 -5377.449,E2 -5377.449} C_VEL
LIN {X 0,Y 509.91,Z 520.967,A -85,B 0,C 180,E1 -5379.844,E2 -5379.844} C_VEL
LIN {X 0,Y 509.881,Z 520.969,A -85,B 0,C 180,E1 -5383.175,E2 -5383.175} C_VEL
LIN {X 0,Y 509.857,Z 520.977,A -85,B 0,C 180,E1 -5385.634,E2 -5385.634} C_VEL
LIN {X 0,Y 509.906,Z 520.963,A -85,B 0,C 180,E1 -5388.874,E2 -5388.874} C_VEL
LIN {X 0,Y 509.945,Z 520.961,A -85,B 0,C 180,E1 -5392.078,E2 -5392.078} C_VEL
LIN {X 0,Y 509.976,Z 520.955,A -85,B 0,C 180,E1 -5394.464,E2 -5394.464} C_VEL
LIN {X 0,Y 510.048,Z 520.951,A -85,B 0,C 180,E1 -5397.631,E2 -5397.631} C_VEL
LIN {X 0,Y 510.058,Z 520.945,A -85,B 0,C 180,E1 -5400.789,E2 -5400.789} C_VEL
LIN {X 0,Y 509.952,Z 520.959,A -85,B 0,C 180,E1 -5403.16,E2 -5403.16} C_VEL
LIN {X 0,Y 509.971,Z 520.956,A -85,B 0,C 180,E1 -5406.33,E2 -5406.33} C_VEL
LIN {X 0,Y 509.909,Z 520.962,A -85,B 0,C 180,E1 -5408.72,E2 -5408.72} C_VEL
LIN {X 0,Y 509.943,Z 520.963,A -85,B 0,C 180,E1 -5411.931,E2 -5411.931} C_VEL
LIN {X 0,Y 509.886,Z 520.969,A -85,B 0,C 180,E1 -5415.242,E2 -5415.242} C_VEL
LIN {X 0,Y 509.881,Z 520.97,A -85,B 0,C 180,E1 -5418.001,E2 -5418.001} C_VEL
LIN {X 0,Y 509.844,Z 520.972,A -85,B 0,C 180,E1 -5421.002,E2 -5421.002} C_VEL
LIN {X 0,Y 509.83,Z 520.98,A -85,B 0,C 180,E1 -5423.564,E2 -5423.564} C_VEL
LIN {X 0,Y 509.907,Z 520.961,A -85,B 0,C 180,E1 -5426.38,E2 -5426.38} C_VEL
LIN {X 0,Y 509.871,Z 520.969,A -85,B 0,C 180,E1 -5428.845,E2 -5428.845} C_VEL
LIN {X 0,Y 509.82,Z 520.981,A -85,B 0,C 180,E1 -5431.59,E2 -5431.59} C_VEL
LIN {X 0,Y 509.849,Z 520.97,A -85,B 0,C 180,E1 -5434.414,E2 -5434.414} C_VEL
LIN {X 0,Y 509.814,Z 520.972,A -85,B 0,C 180,E1 -5437.341,E2 -5437.341} C_VEL
LIN {X 0,Y 509.833,Z 520.974,A -85,B 0,C 180,E1 -5440.383,E2 -5440.383} C_VEL
LIN {X 0,Y 509.819,Z 520.972,A -85,B 0,C 180,E1 -5443.063,E2 -5443.063} C_VEL
LIN {X 0,Y 509.827,Z 520.979,A -85,B 0,C 180,E1 -5445.793,E2 -5445.793} C_VEL
LIN {X 0,Y 509.862,Z 520.97,A -85,B 0,C 180,E1 -5448.576,E2 -5448.576} C_VEL
LIN {X 0,Y 509.849,Z 520.968,A -85,B 0,C 180,E1 -5451.787,E2 -5451.787} C_VEL
LIN {X 0,Y 509.84,Z 520.973,A -85,B 0,C 180,E1 -5454.624,E2 -5454.624} C_VEL
LIN {X 0,Y 509.864,Z 520.959,A -85,B 0,C 180,E1 -5457.482,E2 -5457.482} C_VEL
LIN {X 0,Y 509.857,Z 520.965,A -85,B 0,C 180,E1 -5460.275,E2 -5460.275} C_VEL
LIN {X 0,Y 509.885,Z 520.966,A -85,B 0,C 180,E1 -5462.945,E2 -5462.945} C_VEL
LIN {X 0,Y 509.878,Z 521.07,A -85,B 0,C 180,E1 -5465.399,E2 -5465.399} C_VEL
LIN {X 0,Y 511.388,Z 528.789,A -85,B 0,C 180,E1 -5466.822,E2 -5466.822} C_VEL
LIN {X 0,Y 511.386,Z 535.866,A -85,B 0,C 180,E1 -5468.008,E2 -5468.008} C_VEL
LIN {X 0,Y 510.907,Z 551.117,A -85,B 0,C 180,E1 -5470.515,E2 -5470.515} C_VEL
LIN {X 0,Y 510.459,Z 568.899,A -85,B 0,C 180,E1 -5473.401,E2 -5473.401} C_VEL
LIN {X 0,Y 510.355,Z 575.132,A -85,B 0,C 180,E1 -5474.386,E2 -5474.386} C_VEL
LIN {X 0,Y 510.949,Z 579.363,A -85,B 0,C 180,E1 -5474.499,E2 -5474.499} C_VEL
LIN {X 0,Y 512.269,Z 587.827,A -85,B 0,C 180,E1 -5474.66,E2 -5474.66} C_VEL
LIN {X 0,Y 511.781,Z 683.332,A -85,B 0,C 180,E1 -5476.02,E2 -5476.02} C_VEL
LIN {X 0,Y 511.511,Z 696.597,A -85,B 0,C 180,E1 -5476.367,E2 -5476.367} C_VEL
LIN {X 0,Y 511.208,Z 709.888,A -85,B 0,C 180,E1 -5476.89,E2 -5476.89} C_VEL
LIN {X 0,Y 510.876,Z 722.272,A -85,B 0,C 180,E1 -5477.565,E2 -5477.565} C_VEL
LIN {X 0,Y 510.551,Z 733.95,A -85,B 0,C 180,E1 -5478.387,E2 -5478.387} C_VEL
LIN {X 0,Y 510.181,Z 744.143,A -85,B 0,C 180,E1 -5479.283,E2 -5479.283} C_VEL
LIN {X 0,Y 509.902,Z 753.321,A -85,B 0,C 180,E1 -5480.28,E2 -5480.28} C_VEL
LIN {X 0,Y 509.649,Z 762.264,A -85,B 0,C 180,E1 -5481.476,E2 -5481.476} C_VEL
LIN {X 0,Y 509.436,Z 769.461,A -85,B 0,C 180,E1 -5482.669,E2 -5482.669} C_VEL
LIN {X 0,Y 509.325,Z 774.317,A -85,B 0,C 180,E1 -5483.663,E2 -5483.663} C_VEL
LIN {X 0,Y 509.248,Z 779.039,A -85,B 0,C 180,E1 -5484.854,E2 -5484.854} C_VEL
LIN {X 0,Y 509.25,Z 782.651,A -85,B 0,C 180,E1 -5486.044,E2 -5486.044} C_VEL
LIN {X 0,Y 509.2,Z 784.512,A -85,B 0,C 180,E1 -5486.836,E2 -5486.836} C_VEL
LIN {X 0,Y 509.189,Z 785.906,A -85,B 0,C 180,E1 -5487.628,E2 -5487.628} C_VEL
LIN {X 0,Y 509.073,Z 787.504,A -85,B 0,C 180,E1 -5489.21,E2 -5489.21} C_VEL
LIN {X 0,Y 509.065,Z 787.719,A -85,B 0,C 180,E1 -5490.001,E2 -5490.001} C_VEL
LIN {X 0,Y 509.112,Z 786.895,A -85,B 0,C 180,E1 -5491.583,E2 -5491.583} C_VEL
LIN {X 0,Y 509.189,Z 785.901,A -85,B 0,C 180,E1 -5492.374,E2 -5492.374} C_VEL
LIN {X 0,Y 509.201,Z 784.506,A -85,B 0,C 180,E1 -5493.165,E2 -5493.165} C_VEL
LIN {X 0,Y 509.216,Z 781.573,A -85,B 0,C 180,E1 -5494.354,E2 -5494.354} C_VEL
LIN {X 0,Y 509.322,Z 777.605,A -85,B 0,C 180,E1 -5495.544,E2 -5495.544} C_VEL
LIN {X 0,Y 509.402,Z 771.947,A -85,B 0,C 180,E1 -5496.845,E2 -5496.845} C_VEL
LIN {X 0,Y 509.573,Z 764.815,A -85,B 0,C 180,E1 -5498.128,E2 -5498.128} C_VEL
LIN {X 0,Y 509.794,Z 756.531,A -85,B 0,C 180,E1 -5499.323,E2 -5499.323} C_VEL
LIN {X 0,Y 510.05,Z 748.041,A -85,B 0,C 180,E1 -5500.32,E2 -5500.32} C_VEL
LIN {X 0,Y 510.432,Z 737.552,A -85,B 0,C 180,E1 -5501.316,E2 -5501.316} C_VEL
LIN {X 0,Y 510.716,Z 726.895,A -85,B 0,C 180,E1 -5502.134,E2 -5502.134} C_VEL
LIN {X 0,Y 511.068,Z 715.8,A -85,B 0,C 180,E1 -5502.812,E2 -5502.812} C_VEL
LIN {X 0,Y 511.368,Z 704.139,A -85,B 0,C 180,E1 -5503.36,E2 -5503.36} C_VEL
LIN {X 0,Y 511.629,Z 690.688,A -85,B 0,C 180,E1 -5503.809,E2 -5503.809} C_VEL
LIN {X 0,Y 511.85,Z 677.393,A -85,B 0,C 180,E1 -5504.081,E2 -5504.081} C_VEL
LIN {X 0,Y 512.192,Z 587.159,A -85,B 0,C 180,E1 -5505.352,E2 -5505.352} C_VEL
LIN {X 0,Y 510.374,Z 575.447,A -85,B 0,C 180,E1 -5505.59,E2 -5505.59} C_VEL
LIN {X 0,Y 510.412,Z 571.398,A -85,B 0,C 180,E1 -5506.191,E2 -5506.191} C_VEL
LIN {X 0,Y 510.884,Z 553.65,A -85,B 0,C 180,E1 -5509.07,E2 -5509.07} C_VEL
LIN {X 0,Y 511.44,Z 534.587,A -85,B 0,C 180,E1 -5512.204,E2 -5512.204} C_VEL
LIN {X 0,Y 511.391,Z 528.768,A -85,B 0,C 180,E1 -5513.182,E2 -5513.182} C_VEL
LIN {X 0,Y 509.924,Z 521.23,A -85,B 0,C 180,E1 -5514.544,E2 -5514.544} C_VEL
LIN {X 0,Y 509.881,Z 520.965,A -85,B 0,C 180,E1 -5515.296,E2 -5515.296} C_VEL
LIN {X 0,Y 509.9,Z 520.964,A -85,B 0,C 180,E1 -5518.101,E2 -5518.101} C_VEL
LIN {X 0,Y 509.85,Z 520.973,A -85,B 0,C 180,E1 -5521.28,E2 -5521.28} C_VEL
LIN {X 0,Y 509.86,Z 520.978,A -85,B 0,C 180,E1 -5524.203,E2 -5524.203} C_VEL
LIN {X 0,Y 509.82,Z 520.976,A -85,B 0,C 180,E1 -5527.341,E2 -5527.341} C_VEL
LIN {X 0,Y 509.842,Z 520.979,A -85,B 0,C 180,E1 -5530.382,E2 -5530.382} C_VEL
LIN {X 0,Y 509.828,Z 520.976,A -85,B 0,C 180,E1 -5533.062,E2 -5533.062} C_VEL
LIN {X 0,Y 509.826,Z 520.979,A -85,B 0,C 180,E1 -5535.793,E2 -5535.793} C_VEL
LIN {X 0,Y 509.858,Z 520.975,A -85,B 0,C 180,E1 -5538.575,E2 -5538.575} C_VEL
LIN {X 0,Y 509.855,Z 520.975,A -85,B 0,C 180,E1 -5541.787,E2 -5541.787} C_VEL
LIN {X 0,Y 509.846,Z 520.977,A -85,B 0,C 180,E1 -5544.623,E2 -5544.623} C_VEL
LIN {X 0,Y 509.864,Z 520.972,A -85,B 0,C 180,E1 -5547.481,E2 -5547.481} C_VEL
LIN {X 0,Y 509.862,Z 520.978,A -85,B 0,C 180,E1 -5550.274,E2 -5550.274} C_VEL
LIN {X 0,Y 509.889,Z 520.973,A -85,B 0,C 180,E1 -5552.945,E2 -5552.945} C_VEL
LIN {X 0,Y 509.95,Z 521.248,A -85,B 0,C 180,E1 -5554.325,E2 -5554.325} C_VEL
LIN {X 0,Y 511.507,Z 530.409,A -85,B 0,C 180,E1 -5555.657,E2 -5555.657} C_VEL
LIN {X 0,Y 511.213,Z 553.405,A -85,B 0,C 180,E1 -5558.846,E2 -5558.846} C_VEL
LIN {X 0,Y 510.784,Z 576.088,A -85,B 0,C 180,E1 -5562.025,E2 -5562.025} C_VEL
LIN {X 0,Y 510.466,Z 591.247,A -85,B 0,C 180,E1 -5564.198,E2 -5564.198} C_VEL
LIN {X 0,Y 510.192,Z 606.927,A -85,B 0,C 180,E1 -5566.457,E2 -5566.457} C_VEL
LIN {X 0,Y 510.095,Z 616.711,A -85,B 0,C 180,E1 -5567.789,E2 -5567.789} C_VEL
LIN {X 0,Y 511.053,Z 625.514,A -85,B 0,C 180,E1 -5567.957,E2 -5567.957} C_VEL
LIN {X 0,Y 510.796,Z 696.156,A -85,B 0,C 180,E1 -5568.994,E2 -5568.994} C_VEL
LIN {X 0,Y 510.619,Z 706.961,A -85,B 0,C 180,E1 -5569.292,E2 -5569.292} C_VEL
LIN {X 0,Y 510.429,Z 717.901,A -85,B 0,C 180,E1 -5569.739,E2 -5569.739} C_VEL
LIN {X 0,Y 510.206,Z 729.101,A -85,B 0,C 180,E1 -5570.385,E2 -5570.385} C_VEL
LIN {X 0,Y 509.978,Z 738.281,A -85,B 0,C 180,E1 -5571.081,E2 -5571.081} C_VEL
LIN {X 0,Y 509.754,Z 746.699,A -85,B 0,C 180,E1 -5571.876,E2 -5571.876} C_VEL
LIN {X 0,Y 509.554,Z 754.976,A -85,B 0,C 180,E1 -5572.869,E2 -5572.869} C_VEL
LIN {X 0,Y 509.509,Z 761.493,A -85,B 0,C 180,E1 -5573.863,E2 -5573.863} C_VEL
LIN {X 0,Y 509.286,Z 766.718,A -85,B 0,C 180,E1 -5574.854,E2 -5574.854} C_VEL
LIN {X 0,Y 509.302,Z 771.508,A -85,B 0,C 180,E1 -5576.044,E2 -5576.044} C_VEL
LIN {X 0,Y 509.214,Z 773.892,A -85,B 0,C 180,E1 -5576.835,E2 -5576.835} C_VEL
LIN {X 0,Y 509.191,Z 775.694,A -85,B 0,C 180,E1 -5577.627,E2 -5577.627} C_VEL
LIN {X 0,Y 509.111,Z 776.996,A -85,B 0,C 180,E1 -5578.418,E2 -5578.418} C_VEL
LIN {X 0,Y 509.071,Z 777.798,A -85,B 0,C 180,E1 -5579.209,E2 -5579.209} C_VEL
LIN {X 0,Y 509.064,Z 778.084,A -85,B 0,C 180,E1 -5580,E2 -5580} C_VEL
LIN {X 0,Y 509.072,Z 777.855,A -85,B 0,C 180,E1 -5580.791,E2 -5580.791} C_VEL
LIN {X 0,Y 509.113,Z 777.111,A -85,B 0,C 180,E1 -5581.582,E2 -5581.582} C_VEL
LIN {X 0,Y 509.192,Z 775.866,A -85,B 0,C 180,E1 -5582.373,E2 -5582.373} C_VEL
LIN {X 0,Y 509.249,Z 773.022,A -85,B 0,C 180,E1 -5583.561,E2 -5583.561} C_VEL
LIN {X 0,Y 509.227,Z 768.871,A -85,B 0,C 180,E1 -5584.75,E2 -5584.75} C_VEL
LIN {X 0,Y 509.458,Z 763.167,A -85,B 0,C 180,E1 -5585.939,E2 -5585.939} C_VEL
LIN {X 0,Y 509.529,Z 757.118,A -85,B 0,C 180,E1 -5586.921,E2 -5586.921} C_VEL
LIN {X 0,Y 509.704,Z 749.341,A -85,B 0,C 180,E1 -5587.925,E2 -5587.925} C_VEL
LIN {X 0,Y 509.936,Z 740.536,A -85,B 0,C 180,E1 -5588.82,E2 -5588.82} C_VEL
LIN {X 0,Y 510.183,Z 731.896,A -85,B 0,C 180,E1 -5589.515,E2 -5589.515} C_VEL
LIN {X 0,Y 510.369,Z 722.512,A -85,B 0,C 180,E1 -5590.112,E2 -5590.112} C_VEL
LIN {X 0,Y 510.553,Z 711.097,A -85,B 0,C 180,E1 -5590.66,E2 -5590.66} C_VEL
LIN {X 0,Y 510.699,Z 699.301,A -85,B 0,C 180,E1 -5591.033,E2 -5591.033} C_VEL
LIN {X 0,Y 510.866,Z 685.421,A -85,B 0,C 180,E1 -5591.28,E2 -5591.28} C_VEL
LIN {X 0,Y 511.011,Z 624.58,A -85,B 0,C 180,E1 -5592.151,E2 -5592.151} C_VEL
LIN {X 0,Y 510.066,Z 616.445,A -85,B 0,C 180,E1 -5592.32,E2 -5592.32} C_VEL
LIN {X 0,Y 510.453,Z 594.516,A -85,B 0,C 180,E1 -5595.469,E2 -5595.469} C_VEL
LIN {X 0,Y 510.958,Z 571.169,A -85,B 0,C 180,E1 -5598.859,E2 -5598.859} C_VEL
LIN {X 0,Y 511.424,Z 552.533,A -85,B 0,C 180,E1 -5601.568,E2 -5601.568} C_VEL
LIN {X 0,Y 511.863,Z 533.649,A -85,B 0,C 180,E1 -5604.325,E2 -5604.325} C_VEL
LIN {X 0,Y 511.584,Z 529.514,A -85,B 0,C 180,E1 -5604.948,E2 -5604.948} C_VEL
LIN {X 0,Y 509.919,Z 521.076,A -85,B 0,C 180,E1 -5606.294,E2 -5606.294} C_VEL
LIN {X 0,Y 509.88,Z 520.971,A -85,B 0,C 180,E1 -5608.844,E2 -5608.844} C_VEL
LIN {X 0,Y 509.824,Z 520.983,A -85,B 0,C 180,E1 -5611.59,E2 -5611.59} C_VEL
LIN {X 0,Y 509.855,Z 520.972,A -85,B 0,C 180,E1 -5614.413,E2 -5614.413} C_VEL
LIN {X 0,Y 509.819,Z 520.978,A -85,B 0,C 180,E1 -5617.09,E2 -5617.09} C_VEL
LIN {X 0,Y 509.15,Z 521.066,A -85,B 0,C 180,E1 -5617.749,E2 -5617.749} C_VEL
LIN {X 0,Y 506.287,Z 521.417,A -85,B 0,C 180,E1 -5618.82,E2 -5618.82} C_VEL
LIN {X 0,Y 503.879,Z 521.714,A -85,B 0,C 180,E1 -5619.682,E2 -5619.682} C_VEL
LIN {X 0,Y 502.864,Z 521.835,A -85,B 0,C 180,E1 -5620.348,E2 -5620.348} C_VEL
LIN {X 0,Y 502.791,Z 521.843,A -85,B 0,C 180,E1 -5620.574,E2 -5620.574} C_VEL
LIN {X 0,Y 502.764,Z 521.845,A -85,B 0,C 180,E1 -5623.373,E2 -5623.373} C_VEL
LIN {X 0,Y 502.784,Z 521.856,A -85,B 0,C 180,E1 -5625.66,E2 -5625.66} C_VEL
LIN {X 0,Y 502.823,Z 521.849,A -85,B 0,C 180,E1 -5629.005,E2 -5629.005} C_VEL
LIN {X 0,Y 502.797,Z 521.849,A -85,B 0,C 180,E1 -5632.046,E2 -5632.046} C_VEL
LIN {X 0,Y 502.8,Z 521.854,A -85,B 0,C 180,E1 -5635.034,E2 -5635.034} C_VEL
LIN {X 0,Y 502.787,Z 521.852,A -85,B 0,C 180,E1 -5637.915,E2 -5637.915} C_VEL
LIN {X 0,Y 502.829,Z 521.853,A -85,B 0,C 180,E1 -5640.712,E2 -5640.712} C_VEL
LIN {X 0,Y 502.868,Z 521.845,A -85,B 0,C 180,E1 -5643.439,E2 -5643.439} C_VEL
LIN {X 0,Y 502.782,Z 521.85,A -85,B 0,C 180,E1 -5646.085,E2 -5646.085} C_VEL
LIN {X 0,Y 502.891,Z 522.016,A -85,B 0,C 180,E1 -5648.931,E2 -5648.931} C_VEL
LIN {X 0,Y 503.861,Z 528.027,A -85,B 0,C 180,E1 -5650.229,E2 -5650.229} C_VEL
LIN {X 0,Y 503.455,Z 542.645,A -85,B 0,C 180,E1 -5653.162,E2 -5653.162} C_VEL
LIN {X 0,Y 503.287,Z 548.254,A -85,B 0,C 180,E1 -5654.227,E2 -5654.227} C_VEL
LIN {X 0,Y 504.495,Z 555.05,A -85,B 0,C 180,E1 -5654.397,E2 -5654.397} C_VEL
LIN {X 0,Y 505.432,Z 560.212,A -85,B 0,C 180,E1 -5654.502,E2 -5654.502} C_VEL
LIN {X 0,Y 504.918,Z 655.121,A -85,B 0,C 180,E1 -5655.876,E2 -5655.876} C_VEL
LIN {X 0,Y 504.696,Z 668.29,A -85,B 0,C 180,E1 -5656.229,E2 -5656.229} C_VEL
LIN {X 0,Y 504.403,Z 680.376,A -85,B 0,C 180,E1 -5656.708,E2 -5656.708} C_VEL
LIN {X 0,Y 504.089,Z 692.229,A -85,B 0,C 180,E1 -5657.344,E2 -5657.344} C_VEL
LIN {X 0,Y 503.743,Z 703.44,A -85,B 0,C 180,E1 -5658.124,E2 -5658.124} C_VEL
LIN {X 0,Y 503.354,Z 713.917,A -85,B 0,C 180,E1 -5659.033,E2 -5659.033} C_VEL
LIN {X 0,Y 503.068,Z 722.471,A -85,B 0,C 180,E1 -5659.942,E2 -5659.942} C_VEL
LIN {X 0,Y 502.804,Z 730.351,A -85,B 0,C 180,E1 -5660.952,E2 -5660.952} C_VEL
LIN {X 0,Y 502.52,Z 738.056,A -85,B 0,C 180,E1 -5662.162,E2 -5662.162} C_VEL
LIN {X 0,Y 502.325,Z 745.123,A -85,B 0,C 180,E1 -5663.573,E2 -5663.573} C_VEL
LIN {X 0,Y 502.186,Z 749.833,A -85,B 0,C 180,E1 -5664.78,E2 -5664.78} C_VEL
LIN {X 0,Y 502.235,Z 753.433,A -85,B 0,C 180,E1 -5665.987,E2 -5665.987} C_VEL
LIN {X 0,Y 502.124,Z 755.298,A -85,B 0,C 180,E1 -5666.79,E2 -5666.79} C_VEL
LIN {X 0,Y 502.121,Z 756.705,A -85,B 0,C 180,E1 -5667.593,E2 -5667.593} C_VEL
LIN {X 0,Y 501.991,Z 758.326,A -85,B 0,C 180,E1 -5669.197,E2 -5669.197} C_VEL
LIN {X 0,Y 501.98,Z 758.564,A -85,B 0,C 180,E1 -5669.999,E2 -5669.999} C_VEL
LIN {X 0,Y 501.99,Z 758.381,A -85,B 0,C 180,E1 -5670.801,E2 -5670.801} C_VEL
LIN {X 0,Y 502.121,Z 756.835,A -85,B 0,C 180,E1 -5672.406,E2 -5672.406} C_VEL
LIN {X 0,Y 502.124,Z 755.483,A -85,B 0,C 180,E1 -5673.209,E2 -5673.209} C_VEL
LIN {X 0,Y 502.205,Z 752.619,A -85,B 0,C 180,E1 -5674.414,E2 -5674.414} C_VEL
LIN {X 0,Y 502.288,Z 748.736,A -85,B 0,C 180,E1 -5675.62,E2 -5675.62} C_VEL
LIN {X 0,Y 502.351,Z 743.734,A -85,B 0,C 180,E1 -5676.828,E2 -5676.828} C_VEL
LIN {X 0,Y 502.557,Z 737.432,A -85,B 0,C 180,E1 -5678.038,E2 -5678.038} C_VEL
LIN {X 0,Y 502.782,Z 729.54,A -85,B 0,C 180,E1 -5679.25,E2 -5679.25} C_VEL
LIN {X 0,Y 503.063,Z 721.496,A -85,B 0,C 180,E1 -5680.26,E2 -5680.26} C_VEL
LIN {X 0,Y 503.464,Z 711.675,A -85,B 0,C 180,E1 -5681.269,E2 -5681.269} C_VEL
LIN {X 0,Y 503.856,Z 700.539,A -85,B 0,C 180,E1 -5682.186,E2 -5682.186} C_VEL
LIN {X 0,Y 504.119,Z 689.824,A -85,B 0,C 180,E1 -5682.888,E2 -5682.888} C_VEL
LIN {X 0,Y 504.471,Z 677.867,A -85,B 0,C 180,E1 -5683.494,E2 -5683.494} C_VEL
LIN {X 0,Y 504.761,Z 664.796,A -85,B 0,C 180,E1 -5683.973,E2 -5683.973} C_VEL
LIN {X 0,Y 504.976,Z 651.694,A -85,B 0,C 180,E1 -5684.276,E2 -5684.276} C_VEL
LIN {X 0,Y 505.316,Z 559.485,A -85,B 0,C 180,E1 -5685.603,E2 -5685.603} C_VEL
LIN {X 0,Y 503.3,Z 548.315,A -85,B 0,C 180,E1 -5685.857,E2 -5685.857} C_VEL
LIN {X 0,Y 503.468,Z 542.058,A -85,B 0,C 180,E1 -5687.045,E2 -5687.045} C_VEL
LIN {X 0,Y 503.859,Z 528.475,A -85,B 0,C 180,E1 -5689.769,E2 -5689.769} C_VEL
LIN {X 0,Y 502.869,Z 521.896,A -85,B 0,C 180,E1 -5691.213,E2 -5691.213} C_VEL
LIN {X 0,Y 502.829,Z 521.85,A -85,B 0,C 180,E1 -5694.79,E2 -5694.79} C_VEL
LIN {X 0,Y 502.834,Z 521.853,A -85,B 0,C 180,E1 -5697.466,E2 -5697.466} C_VEL
LIN {X 0,Y 502.809,Z 521.847,A -85,B 0,C 180,E1 -5700.21,E2 -5700.21} C_VEL
LIN {X 0,Y 502.831,Z 521.849,A -85,B 0,C 180,E1 -5703.03,E2 -5703.03} C_VEL
LIN {X 0,Y 502.781,Z 521.852,A -85,B 0,C 180,E1 -5705.949,E2 -5705.949} C_VEL
LIN {X 0,Y 502.8,Z 521.852,A -85,B 0,C 180,E1 -5708.975,E2 -5708.975} C_VEL
LIN {X 0,Y 502.827,Z 521.847,A -85,B 0,C 180,E1 -5712.135,E2 -5712.135} C_VEL
LIN {X 0,Y 502.797,Z 521.852,A -85,B 0,C 180,E1 -5715.467,E2 -5715.467} C_VEL
LIN {X 0,Y 502.822,Z 521.849,A -85,B 0,C 180,E1 -5719.003,E2 -5719.003} C_VEL
LIN {X 0,Y 502.792,Z 521.846,A -85,B 0,C 180,E1 -5722.046,E2 -5722.046} C_VEL
LIN {X 0,Y 502.805,Z 521.852,A -85,B 0,C 180,E1 -5725.034,E2 -5725.034} C_VEL
LIN {X 0,Y 502.783,Z 521.853,A -85,B 0,C 180,E1 -5727.915,E2 -5727.915} C_VEL
LIN {X 0,Y 502.833,Z 521.846,A -85,B 0,C 180,E1 -5730.713,E2 -5730.713} C_VEL
LIN {X 0,Y 502.875,Z 521.845,A -85,B 0,C 180,E1 -5733.434,E2 -5733.434} C_VEL
LIN {X 0,Y 502.785,Z 521.851,A -85,B 0,C 180,E1 -5736.086,E2 -5736.086} C_VEL
LIN {X 0,Y 502.777,Z 521.849,A -85,B 0,C 180,E1 -5738.688,E2 -5738.688} C_VEL
LIN {X 0,Y 502.824,Z 521.851,A -85,B 0,C 180,E1 -5741.248,E2 -5741.248} C_VEL
LIN {X 0,Y 502.817,Z 521.849,A -85,B 0,C 180,E1 -5743.767,E2 -5743.767} C_VEL
LIN {X 0,Y 502.824,Z 521.846,A -85,B 0,C 180,E1 -5746.254,E2 -5746.254} C_VEL
LIN {X 0,Y 502.87,Z 521.839,A -85,B 0,C 180,E1 -5748.717,E2 -5748.717} C_VEL
LIN {X 0,Y 502.895,Z 521.84,A -85,B 0,C 180,E1 -5751.966,E2 -5751.966} C_VEL
LIN {X 0,Y 502.932,Z 521.832,A -85,B 0,C 180,E1 -5754.386,E2 -5754.386} C_VEL
LIN {X 0,Y 503.018,Z 521.826,A -85,B 0,C 180,E1 -5757.598,E2 -5757.598} C_VEL
LIN {X 0,Y 503.019,Z 521.825,A -85,B 0,C 180,E1 -5760,E2 -5760} C_VEL
LIN {X 0,Y 503.018,Z 521.819,A -85,B 0,C 180,E1 -5762.402,E2 -5762.402} C_VEL
LIN {X 0,Y 502.932,Z 521.84,A -85,B 0,C 180,E1 -5765.614,E2 -5765.614} C_VEL
LIN {X 0,Y 502.894,Z 521.839,A -85,B 0,C 180,E1 -5768.033,E2 -5768.033} C_VEL
LIN {X 0,Y 502.885,Z 521.839,A -85,B 0,C 180,E1 -5771.283,E2 -5771.283} C_VEL
LIN {X 0,Y 502.837,Z 521.843,A -85,B 0,C 180,E1 -5774.571,E2 -5774.571} C_VEL
LIN {X 0,Y 502.855,Z 521.847,A -85,B 0,C 180,E1 -5777.907,E2 -5777.907} C_VEL
LIN {X 0,Y 502.821,Z 521.845,A -85,B 0,C 180,E1 -5780.537,E2 -5780.537} C_VEL
LIN {X 0,Y 502.79,Z 521.85,A -85,B 0,C 180,E1 -5783.041,E2 -5783.041} C_VEL
LIN {X 0,Y 502.835,Z 521.85,A -85,B 0,C 180,E1 -5785.676,E2 -5785.676} C_VEL
LIN {X 0,Y 502.834,Z 521.846,A -85,B 0,C 180,E1 -5788.373,E2 -5788.373} C_VEL
LIN {X 0,Y 502.79,Z 521.855,A -85,B 0,C 180,E1 -5791.5,E2 -5791.5} C_VEL
LIN {X 0,Y 502.802,Z 521.848,A -85,B 0,C 180,E1 -5794.446,E2 -5794.446} C_VEL
LIN {X 0,Y 502.776,Z 521.847,A -85,B 0,C 180,E1 -5797.179,E2 -5797.179} C_VEL
LIN {X 0,Y 502.783,Z 521.855,A -85,B 0,C 180,E1 -5800.016,E2 -5800.016} C_VEL
LIN {X 0,Y 502.797,Z 521.847,A -85,B 0,C 180,E1 -5802.2,E2 -5802.2} C_VEL
LIN {X 0,Y 502.797,Z 521.856,A -85,B 0,C 180,E1 -5805.469,E2 -5805.469} C_VEL
LIN {X 0,Y 502.832,Z 521.852,A -85,B 0,C 180,E1 -5807.866,E2 -5807.866} C_VEL
LIN {X 0,Y 502.807,Z 521.847,A -85,B 0,C 180,E1 -5811.026,E2 -5811.026} C_VEL
LIN {X 0,Y 502.781,Z 521.856,A -85,B 0,C 180,E1 -5814.168,E2 -5814.168} C_VEL
LIN {X 0,Y 502.831,Z 521.841,A -85,B 0,C 180,E1 -5816.994,E2 -5816.994} C_VEL
LIN {X 0,Y 502.813,Z 521.834,A -85,B 0,C 180,E1 -5820.066,E2 -5820.066} C_VEL
LIN {X 0,Y 502.833,Z 521.844,A -85,B 0,C 180,E1 -5822.534,E2 -5822.534} C_VEL
LIN {X 0,Y 502.875,Z 521.938,A -85,B 0,C 180,E1 -5825.212,E2 -5825.212} C_VEL
LIN {X 0,Y 504.222,Z 529.089,A -85,B 0,C 180,E1 -5826.555,E2 -5826.555} C_VEL
LIN {X 0,Y 504.589,Z 533.149,A -85,B 0,C 180,E1 -5827.264,E2 -5827.264} C_VEL
LIN {X 0,Y 504.034,Z 549.671,A -85,B 0,C 180,E1 -5830.026,E2 -5830.026} C_VEL
LIN {X 0,Y 503.488,Z 567.438,A -85,B 0,C 180,E1 -5832.955,E2 -5832.955} C_VEL
LIN {X 0,Y 503.327,Z 574.957,A -85,B 0,C 180,E1 -5834.164,E2 -5834.164} C_VEL
LIN {X 0,Y 504.232,Z 580.986,A -85,B 0,C 180,E1 -5834.313,E2 -5834.313} C_VEL
LIN {X 0,Y 505.424,Z 588.47,A -85,B 0,C 180,E1 -5834.459,E2 -5834.459} C_VEL
LIN {X 0,Y 504.892,Z 683.127,A -85,B 0,C 180,E1 -5835.825,E2 -5835.825} C_VEL
LIN {X 0,Y 504.629,Z 696.393,A -85,B 0,C 180,E1 -5836.177,E2 -5836.177} C_VEL
LIN {X 0,Y 504.299,Z 709.684,A -85,B 0,C 180,E1 -5836.707,E2 -5836.707} C_VEL
LIN {X 0,Y 503.93,Z 721.73,A -85,B 0,C 180,E1 -5837.369,E2 -5837.369} C_VEL
LIN {X 0,Y 503.573,Z 733.744,A -85,B 0,C 180,E1 -5838.223,E2 -5838.223} C_VEL
LIN {X 0,Y 503.187,Z 743.938,A -85,B 0,C 180,E1 -5839.132,E2 -5839.132} C_VEL
LIN {X 0,Y 502.877,Z 753.116,A -85,B 0,C 180,E1 -5840.143,E2 -5840.143} C_VEL
LIN {X 0,Y 502.612,Z 762.059,A -85,B 0,C 180,E1 -5841.355,E2 -5841.355} C_VEL
LIN {X 0,Y 502.36,Z 769.256,A -85,B 0,C 180,E1 -5842.565,E2 -5842.565} C_VEL
LIN {X 0,Y 502.235,Z 774.112,A -85,B 0,C 180,E1 -5843.573,E2 -5843.573} C_VEL
LIN {X 0,Y 502.182,Z 778.834,A -85,B 0,C 180,E1 -5844.781,E2 -5844.781} C_VEL
LIN {X 0,Y 502.144,Z 782.446,A -85,B 0,C 180,E1 -5845.988,E2 -5845.988} C_VEL
LIN {X 0,Y 502.12,Z 784.307,A -85,B 0,C 180,E1 -5846.791,E2 -5846.791} C_VEL
LIN {X 0,Y 502.091,Z 785.702,A -85,B 0,C 180,E1 -5847.594,E2 -5847.594} C_VEL
LIN {X 0,Y 501.99,Z 787.3,A -85,B 0,C 180,E1 -5849.199,E2 -5849.199} C_VEL
LIN {X 0,Y 501.98,Z 787.515,A -85,B 0,C 180,E1 -5850.001,E2 -5850.001} C_VEL
LIN {X 0,Y 502.036,Z 786.691,A -85,B 0,C 180,E1 -5851.605,E2 -5851.605} C_VEL
LIN {X 0,Y 502.091,Z 785.697,A -85,B 0,C 180,E1 -5852.407,E2 -5852.407} C_VEL
LIN {X 0,Y 502.121,Z 784.301,A -85,B 0,C 180,E1 -5853.21,E2 -5853.21} C_VEL
LIN {X 0,Y 502.112,Z 781.368,A -85,B 0,C 180,E1 -5854.416,E2 -5854.416} C_VEL
LIN {X 0,Y 502.242,Z 777.399,A -85,B 0,C 180,E1 -5855.622,E2 -5855.622} C_VEL
LIN {X 0,Y 502.333,Z 771.388,A -85,B 0,C 180,E1 -5857.012,E2 -5857.012} C_VEL
LIN {X 0,Y 502.502,Z 764.609,A -85,B 0,C 180,E1 -5858.243,E2 -5858.243} C_VEL
LIN {X 0,Y 502.759,Z 756.326,A -85,B 0,C 180,E1 -5859.454,E2 -5859.454} C_VEL
LIN {X 0,Y 503.033,Z 747.835,A -85,B 0,C 180,E1 -5860.465,E2 -5860.465} C_VEL
LIN {X 0,Y 503.447,Z 737.347,A -85,B 0,C 180,E1 -5861.475,E2 -5861.475} C_VEL
LIN {X 0,Y 503.73,Z 726.689,A -85,B 0,C 180,E1 -5862.305,E2 -5862.305} C_VEL
LIN {X 0,Y 504.122,Z 715.594,A -85,B 0,C 180,E1 -5862.992,E2 -5862.992} C_VEL
LIN {X 0,Y 504.452,Z 703.934,A -85,B 0,C 180,E1 -5863.547,E2 -5863.547} C_VEL
LIN {X 0,Y 504.721,Z 691.4,A -85,B 0,C 180,E1 -5863.976,E2 -5863.976} C_VEL
LIN {X 0,Y 504.941,Z 678.708,A -85,B 0,C 180,E1 -5864.252,E2 -5864.252} C_VEL
LIN {X 0,Y 505.231,Z 586.883,A -85,B 0,C 180,E1 -5865.57,E2 -5865.57} C_VEL
LIN {X 0,Y 503.339,Z 575.13,A -85,B 0,C 180,E1 -5865.821,E2 -5865.821} C_VEL
LIN {X 0,Y 503.862,Z 557.271,A -85,B 0,C 180,E1 -5868.712,E2 -5868.712} C_VEL
LIN {X 0,Y 504.41,Z 538.226,A -85,B 0,C 180,E1 -5871.883,E2 -5871.883} C_VEL
LIN {X 0,Y 504.536,Z 530.632,A -85,B 0,C 180,E1 -5873.167,E2 -5873.167} C_VEL
LIN {X 0,Y 502.875,Z 522.169,A -85,B 0,C 180,E1 -5874.712,E2 -5874.712} C_VEL
LIN {X 0,Y 502.843,Z 521.843,A -85,B 0,C 180,E1 -5875.011,E2 -5875.011} C_VEL
LIN {X 0,Y 502.837,Z 521.849,A -85,B 0,C 180,E1 -5877.467,E2 -5877.467} C_VEL
LIN {X 0,Y 502.813,Z 521.85,A -85,B 0,C 180,E1 -5880.211,E2 -5880.211} C_VEL
LIN {X 0,Y 502.836,Z 521.846,A -85,B 0,C 180,E1 -5883.032,E2 -5883.032} C_VEL
LIN {X 0,Y 502.777,Z 521.857,A -85,B 0,C 180,E1 -5885.951,E2 -5885.951} C_VEL
LIN {X 0,Y 502.805,Z 521.851,A -85,B 0,C 180,E1 -5888.976,E2 -5888.976} C_VEL
LIN {X 0,Y 502.8,Z 521.857,A -85,B 0,C 180,E1 -5892.139,E2 -5892.139} C_VEL
LIN {X 0,Y 502.789,Z 521.853,A -85,B 0,C 180,E1 -5895.47,E2 -5895.47} C_VEL
LIN {X 0,Y 502.823,Z 521.848,A -85,B 0,C 180,E1 -5898.934,E2 -5898.934} C_VEL
LIN {X 0,Y 502.797,Z 521.858,A -85,B 0,C 180,E1 -5902.046,E2 -5902.046} C_VEL
LIN {X 0,Y 502.811,Z 521.85,A -85,B 0,C 180,E1 -5905.035,E2 -5905.035} C_VEL
LIN {X 0,Y 502.787,Z 521.858,A -85,B 0,C 180,E1 -5907.916,E2 -5907.916} C_VEL
LIN {X 0,Y 502.828,Z 521.852,A -85,B 0,C 180,E1 -5910.712,E2 -5910.712} C_VEL
LIN {X 0,Y 502.867,Z 521.85,A -85,B 0,C 180,E1 -5913.881,E2 -5913.881} C_VEL
LIN {X 0,Y 502.931,Z 522.193,A -85,B 0,C 180,E1 -5914.19,E2 -5914.19} C_VEL
LIN {X 0,Y 504.531,Z 531.224,A -85,B 0,C 180,E1 -5915.518,E2 -5915.518} C_VEL
LIN {X 0,Y 504.25,Z 554.338,A -85,B 0,C 180,E1 -5918.754,E2 -5918.754} C_VEL
LIN {X 0,Y 503.772,Z 577.079,A -85,B 0,C 180,E1 -5921.977,E2 -5921.977} C_VEL
LIN {X 0,Y 503.364,Z 598.313,A -85,B 0,C 180,E1 -5925.031,E2 -5925.031} C_VEL
LIN {X 0,Y 503.05,Z 616.571,A -85,B 0,C 180,E1 -5927.611,E2 -5927.611} C_VEL
LIN {X 0,Y 504.093,Z 627.125,A -85,B 0,C 180,E1 -5927.816,E2 -5927.816} C_VEL
LIN {X 0,Y 503.794,Z 696.465,A -85,B 0,C 180,E1 -5928.865,E2 -5928.865} C_VEL
LIN {X 0,Y 503.625,Z 706.432,A -85,B 0,C 180,E1 -5929.141,E2 -5929.141} C_VEL
LIN {X 0,Y 503.44,Z 716.423,A -85,B 0,C 180,E1 -5929.544,E2 -5929.544} C_VEL
LIN {X 0,Y 503.206,Z 727.403,A -85,B 0,C 180,E1 -5930.149,E2 -5930.149} C_VEL
LIN {X 0,Y 502.972,Z 736.931,A -85,B 0,C 180,E1 -5930.854,E2 -5930.854} C_VEL
LIN {X 0,Y 502.773,Z 744.606,A -85,B 0,C 180,E1 -5931.56,E2 -5931.56} C_VEL
LIN {X 0,Y 502.57,Z 751.786,A -85,B 0,C 180,E1 -5932.366,E2 -5932.366} C_VEL
LIN {X 0,Y 502.47,Z 758.763,A -85,B 0,C 180,E1 -5933.327,E2 -5933.327} C_VEL
LIN {X 0,Y 502.314,Z 764.789,A -85,B 0,C 180,E1 -5934.38,E2 -5934.38} C_VEL
LIN {X 0,Y 502.198,Z 770.047,A -85,B 0,C 180,E1 -5935.586,E2 -5935.586} C_VEL
LIN {X 0,Y 502.136,Z 773.915,A -85,B 0,C 180,E1 -5936.791,E2 -5936.791} C_VEL
LIN {X 0,Y 502.094,Z 775.728,A -85,B 0,C 180,E1 -5937.593,E2 -5937.593} C_VEL
LIN {X 0,Y 502.035,Z 777.041,A -85,B 0,C 180,E1 -5938.396,E2 -5938.396} C_VEL
LIN {X 0,Y 501.988,Z 777.854,A -85,B 0,C 180,E1 -5939.198,E2 -5939.198} C_VEL
LIN {X 0,Y 501.978,Z 778.138,A -85,B 0,C 180,E1 -5940,E2 -5940} C_VEL
LIN {X 0,Y 501.989,Z 777.896,A -85,B 0,C 180,E1 -5940.802,E2 -5940.802} C_VEL
LIN {X 0,Y 502.037,Z 777.145,A -85,B 0,C 180,E1 -5941.604,E2 -5941.604} C_VEL
LIN {X 0,Y 502.095,Z 775.904,A -85,B 0,C 180,E1 -5942.407,E2 -5942.407} C_VEL
LIN {X 0,Y 502.174,Z 773.034,A -85,B 0,C 180,E1 -5943.611,E2 -5943.611} C_VEL
LIN {X 0,Y 502.147,Z 768.877,A -85,B 0,C 180,E1 -5944.817,E2 -5944.817} C_VEL
LIN {X 0,Y 502.387,Z 763.135,A -85,B 0,C 180,E1 -5946.023,E2 -5946.023} C_VEL
LIN {X 0,Y 502.455,Z 756.958,A -85,B 0,C 180,E1 -5947.032,E2 -5947.032} C_VEL
LIN {X 0,Y 502.652,Z 749.252,A -85,B 0,C 180,E1 -5948.037,E2 -5948.037} C_VEL
LIN {X 0,Y 502.926,Z 740.391,A -85,B 0,C 180,E1 -5948.944,E2 -5948.944} C_VEL
LIN {X 0,Y 503.158,Z 731.684,A -85,B 0,C 180,E1 -5949.649,E2 -5949.649} C_VEL
LIN {X 0,Y 503.376,Z 722.246,A -85,B 0,C 180,E1 -5950.254,E2 -5950.254} C_VEL
LIN {X 0,Y 503.551,Z 710.721,A -85,B 0,C 180,E1 -5950.81,E2 -5950.81} C_VEL
LIN {X 0,Y 503.72,Z 699.666,A -85,B 0,C 180,E1 -5951.162,E2 -5951.162} C_VEL
LIN {X 0,Y 503.904,Z 687.888,A -85,B 0,C 180,E1 -5951.387,E2 -5951.387} C_VEL
LIN {X 0,Y 503.999,Z 624.719,A -85,B 0,C 180,E1 -5952.317,E2 -5952.317} C_VEL
LIN {X 0,Y 503.025,Z 616.522,A -85,B 0,C 180,E1 -5952.486,E2 -5952.486} C_VEL
LIN {X 0,Y 503.451,Z 596.506,A -85,B 0,C 180,E1 -5955.381,E2 -5955.381} C_VEL
LIN {X 0,Y 503.982,Z 572.349,A -85,B 0,C 180,E1 -5958.918,E2 -5958.918} C_VEL
LIN {X 0,Y 504.485,Z 553.628,A -85,B 0,C 180,E1 -5961.665,E2 -5961.665} C_VEL
LIN {X 0,Y 504.93,Z 534.657,A -85,B 0,C 180,E1 -5964.462,E2 -5964.462} C_VEL
LIN {X 0,Y 504.351,Z 529.187,A -85,B 0,C 180,E1 -5965.298,E2 -5965.298} C_VEL
LIN {X 0,Y 502.885,Z 521.939,A -85,B 0,C 180,E1 -5966.478,E2 -5966.478} C_VEL
LIN {X 0,Y 502.828,Z 521.852,A -85,B 0,C 180,E1 -5969.288,E2 -5969.288} C_VEL
LIN {X 0,Y 502.787,Z 521.856,A -85,B 0,C 180,E1 -5972.085,E2 -5972.085} C_VEL
LIN {X 0,Y 502.808,Z 521.851,A -85,B 0,C 180,E1 -5974.965,E2 -5974.965} C_VEL
LIN {X 0,Y 502.797,Z 521.852,A -85,B 0,C 180,E1 -5977.954,E2 -5977.954} C_VEL
LIN {X 0,Y 502.791,Z 521.843,A -85,B 0,C 180,E1 -5980.574,E2 -5980.574} C_VEL
LIN {X 0,Y 502.149,Z 521.926,A -85,B 0,C 180,E1 -5981.243,E2 -5981.243} C_VEL
LIN {X 0,Y 499.298,Z 522.284,A -85,B 0,C 180,E1 -5982.329,E2 -5982.329} C_VEL
LIN {X 0,Y 496.866,Z 522.587,A -85,B 0,C 180,E1 -5983.204,E2 -5983.204} C_VEL
LIN {X 0,Y 495.813,Z 522.717,A -85,B 0,C 180,E1 -5983.88,E2 -5983.88} C_VEL
LIN {X 0,Y 495.724,Z 522.727,A -85,B 0,C 180,E1 -5984.109,E2 -5984.109} C_VEL
LIN {X 0,Y 495.73,Z 522.737,A -85,B 0,C 180,E1 -5987.117,E2 -5987.117} C_VEL
LIN {X 0,Y 495.76,Z 522.713,A -85,B 0,C 180,E1 -5989.953,E2 -5989.953} C_VEL
LIN {X 0,Y 495.732,Z 522.73,A -85,B 0,C 180,E1 -5992.553,E2 -5992.553} C_VEL
LIN {X 0,Y 495.775,Z 522.727,A -85,B 0,C 180,E1 -5995.456,E2 -5995.456} C_VEL
LIN {X 0,Y 495.759,Z 522.728,A -85,B 0,C 180,E1 -5998.364,E2 -5998.364} C_VEL
LIN {X 0,Y 495.792,Z 522.726,A -85,B 0,C 180,E1 -6001.507,E2 -6001.507} C_VEL
LIN {X 0,Y 495.794,Z 522.724,A -85,B 0,C 180,E1 -6003.932,E2 -6003.932} C_VEL
LIN {X 0,Y 495.764,Z 522.732,A -85,B 0,C 180,E1 -6007.139,E2 -6007.139} C_VEL
LIN {X 0,Y 495.807,Z 522.868,A -85,B 0,C 180,E1 -6008.756,E2 -6008.756} C_VEL
LIN {X 0,Y 496.889,Z 529.235,A -85,B 0,C 180,E1 -6010.156,E2 -6010.156} C_VEL
LIN {X 0,Y 496.465,Z 543.868,A -85,B 0,C 180,E1 -6013.13,E2 -6013.13} C_VEL
LIN {X 0,Y 496.324,Z 548.458,A -85,B 0,C 180,E1 -6014.001,E2 -6014.001} C_VEL
LIN {X 0,Y 497.908,Z 557.202,A -85,B 0,C 180,E1 -6014.213,E2 -6014.213} C_VEL
LIN {X 0,Y 498.621,Z 562.124,A -85,B 0,C 180,E1 -6014.309,E2 -6014.309} C_VEL
LIN {X 0,Y 498.062,Z 655.354,A -85,B 0,C 180,E1 -6015.677,E2 -6015.677} C_VEL
LIN {X 0,Y 497.797,Z 668.514,A -85,B 0,C 180,E1 -6016.034,E2 -6016.034} C_VEL
LIN {X 0,Y 497.509,Z 680.595,A -85,B 0,C 180,E1 -6016.521,E2 -6016.521} C_VEL
LIN {X 0,Y 497.184,Z 691.372,A -85,B 0,C 180,E1 -6017.099,E2 -6017.099} C_VEL
LIN {X 0,Y 496.856,Z 702.366,A -85,B 0,C 180,E1 -6017.853,E2 -6017.853} C_VEL
LIN {X 0,Y 496.406,Z 713.064,A -85,B 0,C 180,E1 -6018.774,E2 -6018.774} C_VEL
LIN {X 0,Y 496.083,Z 722.681,A -85,B 0,C 180,E1 -6019.799,E2 -6019.799} C_VEL
LIN {X 0,Y 495.77,Z 730.561,A -85,B 0,C 180,E1 -6020.823,E2 -6020.823} C_VEL
LIN {X 0,Y 495.495,Z 738.264,A -85,B 0,C 180,E1 -6022.05,E2 -6022.05} C_VEL
LIN {X 0,Y 495.253,Z 745.331,A -85,B 0,C 180,E1 -6023.481,E2 -6023.481} C_VEL
LIN {X 0,Y 495.128,Z 750.04,A -85,B 0,C 180,E1 -6024.706,E2 -6024.706} C_VEL
LIN {X 0,Y 495.15,Z 753.639,A -85,B 0,C 180,E1 -6025.93,E2 -6025.93} C_VEL
LIN {X 0,Y 495.051,Z 755.504,A -85,B 0,C 180,E1 -6026.744,E2 -6026.744} C_VEL
LIN {X 0,Y 495.025,Z 756.91,A -85,B 0,C 180,E1 -6027.558,E2 -6027.558} C_VEL
LIN {X 0,Y 494.911,Z 758.531,A -85,B 0,C 180,E1 -6029.186,E2 -6029.186} C_VEL
LIN {X 0,Y 494.898,Z 758.768,A -85,B 0,C 180,E1 -6029.999,E2 -6029.999} C_VEL
LIN {X 0,Y 494.911,Z 758.585,A -85,B 0,C 180,E1 -6030.813,E2 -6030.813} C_VEL
LIN {X 0,Y 495.025,Z 757.039,A -85,B 0,C 180,E1 -6032.44,E2 -6032.44} C_VEL
LIN {X 0,Y 495.051,Z 755.686,A -85,B 0,C 180,E1 -6033.255,E2 -6033.255} C_VEL
LIN {X 0,Y 495.114,Z 752.822,A -85,B 0,C 180,E1 -6034.477,E2 -6034.477} C_VEL
LIN {X 0,Y 495.234,Z 748.938,A -85,B 0,C 180,E1 -6035.7,E2 -6035.7} C_VEL
LIN {X 0,Y 495.304,Z 743.936,A -85,B 0,C 180,E1 -6036.926,E2 -6036.926} C_VEL
LIN {X 0,Y 495.518,Z 737.633,A -85,B 0,C 180,E1 -6038.153,E2 -6038.153} C_VEL
LIN {X 0,Y 495.776,Z 729.74,A -85,B 0,C 180,E1 -6039.382,E2 -6039.382} C_VEL
LIN {X 0,Y 496.065,Z 721.696,A -85,B 0,C 180,E1 -6040.406,E2 -6040.406} C_VEL
LIN {X 0,Y 496.509,Z 711.873,A -85,B 0,C 180,E1 -6041.429,E2 -6041.429} C_VEL
LIN {X 0,Y 496.872,Z 702.216,A -85,B 0,C 180,E1 -6042.249,E2 -6042.249} C_VEL
LIN {X 0,Y 497.153,Z 691.558,A -85,B 0,C 180,E1 -6042.981,E2 -6042.981} C_VEL
LIN {X 0,Y 497.55,Z 679.185,A -85,B 0,C 180,E1 -6043.633,E2 -6043.633} C_VEL
LIN {X 0,Y 497.867,Z 665.84,A -85,B 0,C 180,E1 -6044.145,E2 -6044.145} C_VEL
LIN {X 0,Y 498.094,Z 653.363,A -85,B 0,C 180,E1 -6044.451,E2 -6044.451} C_VEL
LIN {X 0,Y 498.548,Z 560.697,A -85,B 0,C 180,E1 -6045.805,E2 -6045.805} C_VEL
LIN {X 0,Y 496.33,Z 548.685,A -85,B 0,C 180,E1 -6046.076,E2 -6046.076} C_VEL
LIN {X 0,Y 496.306,Z 547.44,A -85,B 0,C 180,E1 -6046.245,E2 -6046.245} C_VEL
LIN {X 0,Y 496.805,Z 531.762,A -85,B 0,C 180,E1 -6049.416,E2 -6049.416} C_VEL
LIN {X 0,Y 496.689,Z 527.606,A -85,B 0,C 180,E1 -6050.283,E2 -6050.283} C_VEL
LIN {X 0,Y 495.787,Z 522.779,A -85,B 0,C 180,E1 -6051.38,E2 -6051.38} C_VEL
LIN {X 0,Y 495.753,Z 522.73,A -85,B 0,C 180,E1 -6054.274,E2 -6054.274} C_VEL
LIN {X 0,Y 495.814,Z 522.721,A -85,B 0,C 180,E1 -6056.973,E2 -6056.973} C_VEL
LIN {X 0,Y 495.764,Z 522.725,A -85,B 0,C 180,E1 -6060.146,E2 -6060.146} C_VEL
LIN {X 0,Y 495.792,Z 522.727,A -85,B 0,C 180,E1 -6063.244,E2 -6063.244} C_VEL
LIN {X 0,Y 495.726,Z 522.73,A -85,B 0,C 180,E1 -6066.089,E2 -6066.089} C_VEL
LIN {X 0,Y 495.762,Z 522.727,A -85,B 0,C 180,E1 -6068.768,E2 -6068.768} C_VEL
LIN {X 0,Y 495.774,Z 522.729,A -85,B 0,C 180,E1 -6071.778,E2 -6071.778} C_VEL
LIN {X 0,Y 495.745,Z 522.727,A -85,B 0,C 180,E1 -6075.138,E2 -6075.138} C_VEL
LIN {X 0,Y 495.756,Z 522.727,A -85,B 0,C 180,E1 -6078.219,E2 -6078.219} C_VEL
LIN {X 0,Y 495.774,Z 522.723,A -85,B 0,C 180,E1 -6081.229,E2 -6081.229} C_VEL
LIN {X 0,Y 495.753,Z 522.727,A -85,B 0,C 180,E1 -6084.463,E2 -6084.463} C_VEL
LIN {X 0,Y 495.764,Z 522.731,A -85,B 0,C 180,E1 -6087.405,E2 -6087.405} C_VEL
LIN {X 0,Y 495.776,Z 522.725,A -85,B 0,C 180,E1 -6090.254,E2 -6090.254} C_VEL
LIN {X 0,Y 495.827,Z 522.719,A -85,B 0,C 180,E1 -6093.248,E2 -6093.248} C_VEL
LIN {X 0,Y 495.746,Z 522.732,A -85,B 0,C 180,E1 -6095.725,E2 -6095.725} C_VEL
LIN {X 0,Y 495.741,Z 522.725,A -85,B 0,C 180,E1 -6098.371,E2 -6098.371} C_VEL
LIN {X 0,Y 495.778,Z 522.726,A -85,B 0,C 180,E1 -6100.971,E2 -6100.971} C_VEL
LIN {X 0,Y 495.774,Z 522.727,A -85,B 0,C 180,E1 -6103.53,E2 -6103.53} C_VEL
LIN {X 0,Y 495.787,Z 522.724,A -85,B 0,C 180,E1 -6106.055,E2 -6106.055} C_VEL
LIN {X 0,Y 495.844,Z 522.714,A -85,B 0,C 180,E1 -6108.555,E2 -6108.555} C_VEL
LIN {X 0,Y 495.866,Z 522.717,A -85,B 0,C 180,E1 -6111.852,E2 -6111.852} C_VEL
LIN {X 0,Y 495.889,Z 522.71,A -85,B 0,C 180,E1 -6114.306,E2 -6114.306} C_VEL
LIN {X 0,Y 495.987,Z 522.701,A -85,B 0,C 180,E1 -6117.564,E2 -6117.564} C_VEL
LIN {X 0,Y 495.99,Z 522.7,A -85,B 0,C 180,E1 -6120,E2 -6120} C_VEL
LIN {X 0,Y 495.987,Z 522.695,A -85,B 0,C 180,E1 -6122.436,E2 -6122.436} C_VEL
LIN {X 0,Y 495.889,Z 522.717,A -85,B 0,C 180,E1 -6125.694,E2 -6125.694} C_VEL
LIN {X 0,Y 495.865,Z 522.713,A -85,B 0,C 180,E1 -6128.148,E2 -6128.148} C_VEL
LIN {X 0,Y 495.86,Z 522.716,A -85,B 0,C 180,E1 -6131.445,E2 -6131.445} C_VEL
LIN {X 0,Y 495.782,Z 522.722,A -85,B 0,C 180,E1 -6134.783,E2 -6134.783} C_VEL
LIN {X 0,Y 495.781,Z 522.725,A -85,B 0,C 180,E1 -6137.319,E2 -6137.319} C_VEL
LIN {X 0,Y 495.771,Z 522.728,A -85,B 0,C 180,E1 -6139.89,E2 -6139.89} C_VEL
LIN {X 0,Y 495.758,Z 522.725,A -85,B 0,C 180,E1 -6142.863,E2 -6142.863} C_VEL
LIN {X 0,Y 495.793,Z 522.722,A -85,B 0,C 180,E1 -6146.068,E2 -6146.068} C_VEL
LIN {X 0,Y 495.765,Z 522.726,A -85,B 0,C 180,E1 -6148.815,E2 -6148.815} C_VEL
LIN {X 0,Y 495.753,Z 522.734,A -85,B 0,C 180,E1 -6151.727,E2 -6151.727} C_VEL
LIN {X 0,Y 495.772,Z 522.723,A -85,B 0,C 180,E1 -6154.696,E2 -6154.696} C_VEL
LIN {X 0,Y 495.726,Z 522.729,A -85,B 0,C 180,E1 -6157.562,E2 -6157.562} C_VEL
LIN {X 0,Y 495.762,Z 522.726,A -85,B 0,C 180,E1 -6160.701,E2 -6160.701} C_VEL
LIN {X 0,Y 495.729,Z 522.735,A -85,B 0,C 180,E1 -6164.002,E2 -6164.002} C_VEL
LIN {X 0,Y 495.759,Z 522.725,A -85,B 0,C 180,E1 -6167.122,E2 -6167.122} C_VEL
LIN {X 0,Y 495.78,Z 522.722,A -85,B 0,C 180,E1 -6170.366,E2 -6170.366} C_VEL
LIN {X 0,Y 495.73,Z 522.728,A -85,B 0,C 180,E1 -6173.457,E2 -6173.457} C_VEL
LIN {X 0,Y 495.758,Z 522.722,A -85,B 0,C 180,E1 -6176.437,E2 -6176.437} C_VEL
LIN {X 0,Y 495.751,Z 522.699,A -85,B 0,C 180,E1 -6179.314,E2 -6179.314} C_VEL
LIN {X 0,Y 495.78,Z 522.726,A -85,B 0,C 180,E1 -6182.11,E2 -6182.11} C_VEL
LIN {X 0,Y 495.826,Z 522.818,A -85,B 0,C 180,E1 -6185.022,E2 -6185.022} C_VEL
LIN {X 0,Y 497.677,Z 532.975,A -85,B 0,C 180,E1 -6186.93,E2 -6186.93} C_VEL
LIN {X 0,Y 497.13,Z 549.497,A -85,B 0,C 180,E1 -6189.736,E2 -6189.736} C_VEL
LIN {X 0,Y 496.487,Z 568.502,A -85,B 0,C 180,E1 -6192.92,E2 -6192.92} C_VEL
LIN {X 0,Y 496.328,Z 574.826,A -85,B 0,C 180,E1 -6193.94,E2 -6193.94} C_VEL
LIN {X 0,Y 497.618,Z 583.215,A -85,B 0,C 180,E1 -6194.135,E2 -6194.135} C_VEL
LIN {X 0,Y 498.57,Z 590.095,A -85,B 0,C 180,E1 -6194.267,E2 -6194.267} C_VEL
LIN {X 0,Y 498.015,Z 682.923,A -85,B 0,C 180,E1 -6195.625,E2 -6195.625} C_VEL
LIN {X 0,Y 497.742,Z 696.188,A -85,B 0,C 180,E1 -6195.982,E2 -6195.982} C_VEL
LIN {X 0,Y 497.413,Z 708.356,A -85,B 0,C 180,E1 -6196.467,E2 -6196.467} C_VEL
LIN {X 0,Y 497.039,Z 720.483,A -85,B 0,C 180,E1 -6197.123,E2 -6197.123} C_VEL
LIN {X 0,Y 496.618,Z 732.243,A -85,B 0,C 180,E1 -6197.952,E2 -6197.952} C_VEL
LIN {X 0,Y 496.254,Z 742.688,A -85,B 0,C 180,E1 -6198.875,E2 -6198.875} C_VEL
LIN {X 0,Y 495.894,Z 751.23,A -85,B 0,C 180,E1 -6199.797,E2 -6199.797} C_VEL
LIN {X 0,Y 495.632,Z 759.112,A -85,B 0,C 180,E1 -6200.822,E2 -6200.822} C_VEL
LIN {X 0,Y 495.375,Z 766.811,A -85,B 0,C 180,E1 -6202.05,E2 -6202.05} C_VEL
LIN {X 0,Y 495.163,Z 773.906,A -85,B 0,C 180,E1 -6203.481,E2 -6203.481} C_VEL
LIN {X 0,Y 495.118,Z 778.63,A -85,B 0,C 180,E1 -6204.707,E2 -6204.707} C_VEL
LIN {X 0,Y 495.038,Z 782.24,A -85,B 0,C 180,E1 -6205.93,E2 -6205.93} C_VEL
LIN {X 0,Y 495.042,Z 784.103,A -85,B 0,C 180,E1 -6206.745,E2 -6206.745} C_VEL
LIN {X 0,Y 494.997,Z 785.497,A -85,B 0,C 180,E1 -6207.56,E2 -6207.56} C_VEL
LIN {X 0,Y 494.962,Z 786.49,A -85,B 0,C 180,E1 -6208.373,E2 -6208.373} C_VEL
LIN {X 0,Y 494.898,Z 787.311,A -85,B 0,C 180,E1 -6210.001,E2 -6210.001} C_VEL
LIN {X 0,Y 494.962,Z 786.487,A -85,B 0,C 180,E1 -6211.628,E2 -6211.628} C_VEL
LIN {X 0,Y 494.998,Z 785.492,A -85,B 0,C 180,E1 -6212.442,E2 -6212.442} C_VEL
LIN {X 0,Y 495.042,Z 784.097,A -85,B 0,C 180,E1 -6213.256,E2 -6213.256} C_VEL
LIN {X 0,Y 495.016,Z 781.162,A -85,B 0,C 180,E1 -6214.479,E2 -6214.479} C_VEL
LIN {X 0,Y 495.16,Z 777.194,A -85,B 0,C 180,E1 -6215.703,E2 -6215.703} C_VEL
LIN {X 0,Y 495.258,Z 771.081,A -85,B 0,C 180,E1 -6217.133,E2 -6217.133} C_VEL
LIN {X 0,Y 495.447,Z 764.404,A -85,B 0,C 180,E1 -6218.361,E2 -6218.361} C_VEL
LIN {X 0,Y 495.731,Z 756.12,A -85,B 0,C 180,E1 -6219.59,E2 -6219.59} C_VEL
LIN {X 0,Y 496.014,Z 747.629,A -85,B 0,C 180,E1 -6220.615,E2 -6220.615} C_VEL
LIN {X 0,Y 496.474,Z 737.141,A -85,B 0,C 180,E1 -6221.638,E2 -6221.638} C_VEL
LIN {X 0,Y 496.789,Z 725.619,A -85,B 0,C 180,E1 -6222.542,E2 -6222.542} C_VEL
LIN {X 0,Y 497.224,Z 713.465,A -85,B 0,C 180,E1 -6223.279,E2 -6223.279} C_VEL
LIN {X 0,Y 497.61,Z 701.124,A -85,B 0,C 180,E1 -6223.841,E2 -6223.841} C_VEL
LIN {X 0,Y 497.924,Z 688.447,A -85,B 0,C 180,E1 -6224.249,E2 -6224.249} C_VEL
LIN {X 0,Y 498.137,Z 675.206,A -85,B 0,C 180,E1 -6224.503,E2 -6224.503} C_VEL
LIN {X 0,Y 498.424,Z 587.892,A -85,B 0,C 180,E1 -6225.77,E2 -6225.77} C_VEL
LIN {X 0,Y 496.382,Z 575.249,A -85,B 0,C 180,E1 -6226.032,E2 -6226.032} C_VEL
LIN {X 0,Y 496.364,Z 573.526,A -85,B 0,C 180,E1 -6226.242,E2 -6226.242} C_VEL
LIN {X 0,Y 496.916,Z 555.83,A -85,B 0,C 180,E1 -6229.198,E2 -6229.198} C_VEL
LIN {X 0,Y 497.585,Z 536.779,A -85,B 0,C 180,E1 -6232.418,E2 -6232.418} C_VEL
LIN {X 0,Y 497.485,Z 531.541,A -85,B 0,C 180,E1 -6233.327,E2 -6233.327} C_VEL
LIN {X 0,Y 495.83,Z 522.813,A -85,B 0,C 180,E1 -6234.979,E2 -6234.979} C_VEL
LIN {X 0,Y 495.785,Z 522.724,A -85,B 0,C 180,E1 -6237.892,E2 -6237.892} C_VEL
LIN {X 0,Y 495.756,Z 522.732,A -85,B 0,C 180,E1 -6240.688,E2 -6240.688} C_VEL
LIN {X 0,Y 495.763,Z 522.728,A -85,B 0,C 180,E1 -6243.565,E2 -6243.565} C_VEL
LIN {X 0,Y 495.732,Z 522.735,A -85,B 0,C 180,E1 -6246.544,E2 -6246.544} C_VEL
LIN {X 0,Y 495.76,Z 522.729,A -85,B 0,C 180,E1 -6249.638,E2 -6249.638} C_VEL
LIN {X 0,Y 495.741,Z 522.735,A -85,B 0,C 180,E1 -6252.507,E2 -6252.507} C_VEL
LIN {X 0,Y 495.741,Z 522.731,A -85,B 0,C 180,E1 -6255.141,E2 -6255.141} C_VEL
LIN {X 0,Y 495.759,Z 522.734,A -85,B 0,C 180,E1 -6258.219,E2 -6258.219} C_VEL
LIN {X 0,Y 495.754,Z 522.729,A -85,B 0,C 180,E1 -6261.409,E2 -6261.409} C_VEL
LIN {X 0,Y 495.759,Z 522.733,A -85,B 0,C 180,E1 -6264.463,E2 -6264.463} C_VEL
LIN {X 0,Y 495.771,Z 522.728,A -85,B 0,C 180,E1 -6267.406,E2 -6267.406} C_VEL
LIN {X 0,Y 495.77,Z 522.734,A -85,B 0,C 180,E1 -6270.254,E2 -6270.254} C_VEL
LIN {X 0,Y 495.827,Z 522.725,A -85,B 0,C 180,E1 -6273.251,E2 -6273.251} C_VEL
LIN {X 0,Y 495.858,Z 522.914,A -85,B 0,C 180,E1 -6273.992,E2 -6273.992} C_VEL
LIN {X 0,Y 497.546,Z 532.108,A -85,B 0,C 180,E1 -6275.374,E2 -6275.374} C_VEL
LIN {X 0,Y 497.348,Z 549.253,A -85,B 0,C 180,E1 -6277.79,E2 -6277.79} C_VEL
LIN {X 0,Y 496.968,Z 567.37,A -85,B 0,C 180,E1 -6280.375,E2 -6280.375} C_VEL
LIN {X 0,Y 496.596,Z 585.156,A -85,B 0,C 180,E1 -6282.923,E2 -6282.923} C_VEL
LIN {X 0,Y 496.224,Z 604.051,A -85,B 0,C 180,E1 -6285.65,E2 -6285.65} C_VEL
LIN {X 0,Y 496.028,Z 616.496,A -85,B 0,C 180,E1 -6287.429,E2 -6287.429} C_VEL
LIN {X 0,Y 497.149,Z 627.116,A -85,B 0,C 180,E1 -6287.648,E2 -6287.648} C_VEL
LIN {X 0,Y 496.847,Z 695.707,A -85,B 0,C 180,E1 -6288.707,E2 -6288.707} C_VEL
LIN {X 0,Y 496.651,Z 705.912,A -85,B 0,C 180,E1 -6288.987,E2 -6288.987} C_VEL
LIN {X 0,Y 496.514,Z 714.935,A -85,B 0,C 180,E1 -6289.345,E2 -6289.345} C_VEL
LIN {X 0,Y 496.332,Z 723.727,A -85,B 0,C 180,E1 -6289.805,E2 -6289.805} C_VEL
LIN {X 0,Y 496.084,Z 732.912,A -85,B 0,C 180,E1 -6290.418,E2 -6290.418} C_VEL
LIN {X 0,Y 495.826,Z 742.502,A -85,B 0,C 180,E1 -6291.235,E2 -6291.235} C_VEL
LIN {X 0,Y 495.57,Z 750.044,A -85,B 0,C 180,E1 -6292.052,E2 -6292.052} C_VEL
LIN {X 0,Y 495.397,Z 756.821,A -85,B 0,C 180,E1 -6292.952,E2 -6292.952} C_VEL
LIN {X 0,Y 495.345,Z 762.577,A -85,B 0,C 180,E1 -6293.892,E2 -6293.892} C_VEL
LIN {X 0,Y 495.161,Z 766.681,A -85,B 0,C 180,E1 -6294.707,E2 -6294.707} C_VEL
LIN {X 0,Y 495.095,Z 770.054,A -85,B 0,C 180,E1 -6295.522,E2 -6295.522} C_VEL
LIN {X 0,Y 495.061,Z 773.931,A -85,B 0,C 180,E1 -6296.745,E2 -6296.745} C_VEL
LIN {X 0,Y 495.001,Z 775.759,A -85,B 0,C 180,E1 -6297.559,E2 -6297.559} C_VEL
LIN {X 0,Y 494.961,Z 777.077,A -85,B 0,C 180,E1 -6298.373,E2 -6298.373} C_VEL
LIN {X 0,Y 494.908,Z 777.902,A -85,B 0,C 180,E1 -6299.186,E2 -6299.186} C_VEL
LIN {X 0,Y 494.896,Z 778.193,A -85,B 0,C 180,E1 -6300,E2 -6300} C_VEL
LIN {X 0,Y 494.91,Z 777.936,A -85,B 0,C 180,E1 -6300.814,E2 -6300.814} C_VEL
LIN {X 0,Y 494.963,Z 777.179,A -85,B 0,C 180,E1 -6301.627,E2 -6301.627} C_VEL
LIN {X 0,Y 495.001,Z 775.932,A -85,B 0,C 180,E1 -6302.441,E2 -6302.441} C_VEL
LIN {X 0,Y 495.099,Z 773.046,A -85,B 0,C 180,E1 -6303.662,E2 -6303.662} C_VEL
LIN {X 0,Y 495.072,Z 768.882,A -85,B 0,C 180,E1 -6304.886,E2 -6304.886} C_VEL
LIN {X 0,Y 495.32,Z 763.101,A -85,B 0,C 180,E1 -6306.109,E2 -6306.109} C_VEL
LIN {X 0,Y 495.393,Z 757.043,A -85,B 0,C 180,E1 -6307.11,E2 -6307.11} C_VEL
LIN {X 0,Y 495.566,Z 750.813,A -85,B 0,C 180,E1 -6307.948,E2 -6307.948} C_VEL
LIN {X 0,Y 495.802,Z 742.443,A -85,B 0,C 180,E1 -6308.868,E2 -6308.868} C_VEL
LIN {X 0,Y 496.124,Z 732.89,A -85,B 0,C 180,E1 -6309.684,E2 -6309.684} C_VEL
LIN {X 0,Y 496.354,Z 723.722,A -85,B 0,C 180,E1 -6310.298,E2 -6310.298} C_VEL
LIN {X 0,Y 496.533,Z 713.864,A -85,B 0,C 180,E1 -6310.809,E2 -6310.809} C_VEL
LIN {X 0,Y 496.716,Z 702.091,A -85,B 0,C 180,E1 -6311.244,E2 -6311.244} C_VEL
LIN {X 0,Y 496.9,Z 690.497,A -85,B 0,C 180,E1 -6311.495,E2 -6311.495} C_VEL
LIN {X 0,Y 497.102,Z 625.681,A -85,B 0,C 180,E1 -6312.472,E2 -6312.472} C_VEL
LIN {X 0,Y 496.021,Z 616.485,A -85,B 0,C 180,E1 -6312.665,E2 -6312.665} C_VEL
LIN {X 0,Y 496.467,Z 595.607,A -85,B 0,C 180,E1 -6315.716,E2 -6315.716} C_VEL
LIN {X 0,Y 497.062,Z 572.076,A -85,B 0,C 180,E1 -6319.192,E2 -6319.192} C_VEL
LIN {X 0,Y 497.622,Z 550.331,A -85,B 0,C 180,E1 -6322.416,E2 -6322.416} C_VEL
LIN {X 0,Y 498.013,Z 535.639,A -85,B 0,C 180,E1 -6324.602,E2 -6324.602} C_VEL
LIN {X 0,Y 497.12,Z 529.327,A -85,B 0,C 180,E1 -6325.591,E2 -6325.591} C_VEL
LIN {X 0,Y 495.849,Z 522.804,A -85,B 0,C 180,E1 -6326.667,E2 -6326.667} C_VEL
LIN {X 0,Y 495.77,Z 522.733,A -85,B 0,C 180,E1 -6329.746,E2 -6329.746} C_VEL
LIN {X 0,Y 495.771,Z 522.727,A -85,B 0,C 180,E1 -6332.594,E2 -6332.594} C_VEL
LIN {X 0,Y 495.755,Z 522.735,A -85,B 0,C 180,E1 -6335.537,E2 -6335.537} C_VEL
LIN {X 0,Y 495.767,Z 522.725,A -85,B 0,C 180,E1 -6338.768,E2 -6338.768} C_VEL
LIN {X 0,Y 495.759,Z 522.711,A -85,B 0,C 180,E1 -6341.781,E2 -6341.781} C_VEL
LIN {X 0,Y 495.724,Z 522.727,A -85,B 0,C 180,E1 -6344.109,E2 -6344.109} C_VEL
LIN {X 0,Y 495.051,Z 522.812,A -85,B 0,C 180,E1 -6344.787,E2 -6344.787} C_VEL
LIN {X 0,Y 492.206,Z 523.172,A -85,B 0,C 180,E1 -6345.889,E2 -6345.889} C_VEL
LIN {X 0,Y 489.805,Z 523.474,A -85,B 0,C 180,E1 -6346.776,E2 -6346.776} C_VEL
LIN {X 0,Y 488.773,Z 523.602,A -85,B 0,C 180,E1 -6347.462,E2 -6347.462} C_VEL
LIN {X 0,Y 488.688,Z 523.608,A -85,B 0,C 180,E1 -6347.694,E2 -6347.694} C_VEL
LIN {X 0,Y 488.702,Z 523.594,A -85,B 0,C 180,E1 -6350.745,E2 -6350.745} C_VEL
